// TwinCAT 3 PLC project PRG_B_Base
// Title: B_Base
// Company: RafalOS
// Author: Rafał Osajda
// ProjectVersion: 0.0.1.0
// ProgramVersion: 3.1.4024.0
// libraries:
//   Tc2_Standard, * (Beckhoff Automation GmbH)
//   Tc2_System, * (Beckhoff Automation GmbH)
//   Tc2_Utilities, * (Beckhoff Automation GmbH)
//   Tc3_Module, * (Beckhoff Automation GmbH)
// project tree:
//   DUTs Events/ E_BaseEvents_Category.TcDUT, E_BaseEvents_Action.TcDUT (not stored), ST_BaseEvents.TcDUT (not stored), ST_BaseEvents_ActiveEvents.TcDUT (not stored), ST_BaseEvents_Definition.TcDUT, ST_BaseEvents_Queue.TcDUT, ST_BaseEvents_Memory.TcDUT, ST_BaseEvents_RowInQueue.TcDUT (not stored), ST_BaseEvents_RowInMemory.TcDUT (not stored), ST_BaseEvents_InformationAboutEventsForHMI.TcDUT
//   DUTs/ E_BaseElementType.TcDUT (not stored), E_BaseLocation.TcDUT (not stored), E_BaseMachineState.TcDUT (not stored), E_BaseMachineMode.TcDUT (not stored), ST_BaseCommonData.TcDUT, ST_BaseDescriptor.TcDUT, ST_BaseElementIdentifier.TcDUT (not stored), ST_BaseLocationDesctription.TcDUT, ST_BaseLabel.TcDUT
//   FUNs/ CreateElementCode.TcPOU
//   GVLs/ GVL_BaseConstans.TcGVL (not stored)
//   ITFs/ ITF_DecoratedElement.TcIO (not stored)
//   / PlcTask.TcTTO
//   POUs Compilation/ PRG_Compilation.TcPOU
//   POUs/A01_Base/ ITF_Base.TcIO, FB_Base.TcPOU (not stored)
//   POUs/A02_FB_BaseLogger/ ITF_BaseLogger_HMI_Connector.TcIO, ITF_BaseLogger_HMI_Connector_Command.TcIO, FB_BaseLogger.TcPOU (not stored), ITF_BaseLogger.TcIO, ITF_BaseLogger_HMI_Connector_View.TcIO, ITF_BaseLogger_Item.TcIO, ST_BaseLogger_ItemDataToDisplay.TcDUT
//   POUs/A03_FB_BaseLoggerElement/ ITF_BaseLoggerElement_HMI_Connector.TcIO, ITF_BaseLoggerElement_HMI_Connector_Command.TcIO, FB_BaseLoggerElement.TcPOU, ITF_BaseLoggerElement.TcIO, ITF_BaseLoggerElement_HMI_Connector_View.TcIO
//   POUs/A04_FB_BaseComponent/ ITF_BaseComponent_HMI_Connector.TcIO, ITF_BaseComponent_HMI_Connector_Command.TcIO, FB_BaseComponent.TcPOU, ITF_BaseComponent.TcIO, ITF_BaseComponent_HMI_Connector_View.TcIO, ST_Parameters.TcDUT
//   POUs/A05_FB_BaseControlElement/ ITF_BaseControlElement_HMI_Connector.TcIO, ITF_BaseControlElement_HMI_Connector_Command.TcIO, FB_BaseControlElement.TcPOU, ITF_BaseControlElement.TcIO, ITF_BaseControlElement_HMI_Connector_View.TcIO, ST_BaseControlElement_Power.TcDUT, ST_BaseControlElement_Homing.TcDUT (not stored)
//   POUs/A06_FB_BaseGroupElement/ ITF_BaseGroupElement_HMI_Connector.TcIO, ITF_BaseGroupElement_HMI_Connector_Command.TcIO, FB_BaseGroupElement.TcPOU, ITF_BaseGroupElement.TcIO (not stored), ITF_BaseGroupElement_HMI_Connector_View.TcIO
//   POUs/A07_FB_BaseTopElement/ ITF_BaseSaM.TcIO, ITF_BaseSaMStateMethod.TcIO (not stored), ITF_BaseTopElement_HMI_Connector.TcIO, ITF_BaseTopElement_HMI_Connector_Command.TcIO, FB_BaseTopElement.TcPOU (not stored), ITF_BaseTopElement.TcIO (not stored), ITF_BaseTopElement_HMI_Connector_View.TcIO
//   POUs/B01_Komunikator/ ITF_BaseCommunicator.TcIO, ITF_BaseMessengerRecipient.TcIO, ITF_BaseMessengerSender.TcIO (not stored), FB_BaseCommunicator.TcPOU (not stored), ST_BaseCommunicatorData.TcDUT, ST_BaseCommunicatorStack.TcDUT, ST_BaseCommunicatorMassege.TcDUT (not stored)
//   POUs/B02_Recipes/ FB_BaseRecipe.TcPOU, ITF_BaseCreateTemplateOfRecipe.TcIO (not stored), ITF_BaseCreatingTemplateMethod.TcIO, ITF_BaseRecipe.TcIO, ITF_BaseRecipe_HMI_Connector.TcIO, ST_BaseRecipeListRow.TcDUT, ST_BaseRecipe.TcDUT (not stored), ST_BaseRecipeList.TcDUT
//   POUs/A00_Basic/ FB_BaseLabel.TcPOU, FB_BaseTime.TcPOU (not stored), FB_BaseCommand.TcPOU (not stored), FB_BaseDescriptor.TcPOU, FB_BaseFlag.TcPOU, FB_BaseImpulse.TcPOU (not stored), FB_BaseLocation.TcPOU (not stored), ITF_BaseDescriptor.TcIO, ITF_BaseFlag.TcIO (not stored), ITF_BaseFlagGet.TcIO, ITF_BaseFlagSet.TcIO (not stored), ITF_BaseImpulse.TcIO (not stored), ITF_BaseLabel.TcIO, ITF_BaseLocation.TcIO, ITF_BaseTime.TcIO

CONFIGURATION PRG_B_Base
    RESOURCE PLC ON TwinCAT3
        TASK PlcTask(INTERVAL := T#10ms, PRIORITY := 20);
        PROGRAM PRG_Compilation WITH PlcTask : PRG_Compilation;
    END_RESOURCE
END_CONFIGURATION

// ---- DUTs Events/E_BaseEvents_Category.TcDUT
{attribute 'qualified_only'}
{attribute 'strict'}
{attribute 'to_string'}
TYPE E_BaseEvents_Category :
(
	None		:= 0,
	Error		:= 1, 
	Alarm		:= 2, 
	Safety		:= 3, 
	Message		:= 4

);
END_TYPE

// ---- DUTs Events/ST_BaseEvents_Definition.TcDUT
TYPE ST_BaseEvents_Definition :
STRUCT
	uiIDEvent								: UINT;						//unikalny numer zgloszenia dla całego projektu nadawany automatycznie 
	uiIDInItem								: UINT;						//unikalny numer w elemencie - ustawiany podczas dodawania zgłoszenia DO elementu
	bIgnoreRepetitions						: BOOL;						//jak true nie zliczaj powtorzeń wystapienia np komunikaty - alarmy 
	uiRepetitionCounter						: UINT;						//licznik powtórzeń po którym ma się zgłosic błąd
	eEventCategory							: E_BaseEvents_Category;	//BYTE;	//1 - blad, 2 - ostrzezenie, 3 - wiadomosc, 4 - safety
	stDescription							: ST_BaseLabel;
	bConfirm								: BOOL;						// w przypadków niektórych zgłoszeń żeby błąd został skasowany należy go zatwierdzić że operator go zobaczył
END_STRUCT
END_TYPE

// ---- DUTs Events/ST_BaseEvents_Queue.TcDUT
TYPE ST_BaseEvents_Queue :
STRUCT
	arrEvents						: ARRAY [1..GVL_BaseConstans.MAX_NUMBER_OF_EVENTS_IN_THE_QUEUE] OF ST_BaseEvents_RowInQueue;
	iNumerOfEvents					: INT;

END_STRUCT
END_TYPE

// ---- DUTs Events/ST_BaseEvents_Memory.TcDUT
TYPE ST_BaseEvents_Memory :
STRUCT
	arrRow						: ARRAY [1..GVL_BaseConstans.MAX_EVENTS_IN_MEMORY] OF ST_BaseEvents_RowInMemory;
	iNumberOfRow				: INT;
	
END_STRUCT
END_TYPE

// ---- DUTs Events/ST_BaseEvents_InformationAboutEventsForHMI.TcDUT
(*			
	RafalOS
	Rafał Osajda		03.09.2025		TC 4024.66
	Informacja czy w danym elemencie jest jakieś nowe zgłoszenie jeszcze nei wyświetlane i ilosc zgloszen calkowita
*)
TYPE ST_BaseEvents_InformationAboutEventsForHMI :
STRUCT
	bNew				: BOOL;	//nowe
	iQuantity			: INT;	//Ilość
END_STRUCT
END_TYPE

// ---- DUTs/ST_BaseCommonData.TcDUT
TYPE ST_BaseCommonData :
STRUCT
	itfLogger				: ITF_BaseLogger;
	itfTime					: ITF_BaseTime;
	itfLocaciotn			: ITF_BaseLocation;
END_STRUCT
END_TYPE

// ---- DUTs/ST_BaseDescriptor.TcDUT
TYPE ST_BaseDescriptor :
STRUCT
	stTexts						: ST_BaseLabel;
	sUnit						: STRING(6);
	rValue						: REAL;
	rMin						: REAL;
	rMax						: REAL;
	rDefaultValue				: REAL;
	
END_STRUCT
END_TYPE

// ---- DUTs/ST_BaseLocationDesctription.TcDUT
TYPE ST_BaseLocationDesctription :
STRUCT
	wsDescription		: WSTRING;
	sCode				: STRING(5);
END_STRUCT
END_TYPE

// ---- DUTs/ST_BaseLabel.TcDUT
TYPE ST_BaseLabel :
STRUCT
	arrText		: ARRAY [1..GVL_BaseConstans.NUMBER_OF_LOCATIONS] OF WSTRING;
	
END_STRUCT
END_TYPE

// ---- POUs/B01_Komunikator/ST_BaseCommunicatorData.TcDUT
TYPE ST_BaseCommunicatorData :
STRUCT
	stMessage					: ST_BaseCommunicatorMassege;
	itfSender					: ITF_BaseMessengerSender;
	arritfRecipient				: ARRAY [1..GVL_BaseConstans.MAX_NUMBER_OF_CLIENTS] OF ITF_BaseMessengerRecipient;
	arrConfirmations			: ARRAY [1..GVL_BaseConstans.MAX_NUMBER_OF_CLIENTS] OF BOOL;		//potwierdzenia
	iNumberOfConfirmations		: INT;	//ilosc odbiorcow ktorzy musza potwierdzic
	iNumberOfRecipient			: INT;
END_STRUCT
END_TYPE

// ---- POUs/B01_Komunikator/ST_BaseCommunicatorStack.TcDUT
TYPE ST_BaseCommunicatorStack :
STRUCT
	stMessage					: ST_BaseCommunicatorMassege;
	bSent						: BOOL;		//wysłane
	bConfirmation				: BOOL;		//potwierdzenie
	itfSender					: ITF_BaseMessengerSender;
	itfRecipient				: ITF_BaseMessengerRecipient;
	
END_STRUCT
END_TYPE

// ---- POUs/A02_FB_BaseLogger/ST_BaseLogger_ItemDataToDisplay.TcDUT
TYPE ST_BaseLogger_ItemDataToDisplay :
STRUCT
	sCode						: STRING;
	sEventCategory				: STRING;
	eEventCategory				: E_BaseEvents_Category;
	stDescription				: ST_BaseLabel;
	stItemName					: ST_BaseLabel;
	uiRepetitionCounter			: UINT;
END_STRUCT
END_TYPE

// ---- POUs/A04_FB_BaseComponent/ST_Parameters.TcDUT
TYPE ST_Parameters :
STRUCT
	arrRow	 				: ARRAY [1..GVL_BaseConstans.MAX_NUMBER_OF_PARAMETERS] OF ST_BaseDescriptor;
	uiNumber				: UINT;
END_STRUCT
END_TYPE

// ---- POUs/A05_FB_BaseControlElement/ST_BaseControlElement_Power.TcDUT
TYPE ST_BaseControlElement_Power :
STRUCT
	cmdTurnOn				: FB_BaseCommand;
	cmdTurnOff				: FB_BaseCommand;
	bStatus					: BOOL;
END_STRUCT
END_TYPE

// ---- POUs/B02_Recipes/ST_BaseRecipeListRow.TcDUT
TYPE ST_BaseRecipeListRow :
STRUCT
	wsText			: WSTRING;
	iNumber			: INT;
	refRecipe		: REFERENCE TO ST_BaseRecipe;
END_STRUCT
END_TYPE

// ---- POUs/B02_Recipes/ST_BaseRecipeList.TcDUT
TYPE ST_BaseRecipeList :
STRUCT
	arrName 	: ARRAY [1..GVL_BaseConstans.MAX_NUMBER_OF_RECIPES] OF ST_BaseLabel;
	iNumber		: INT;
END_STRUCT
END_TYPE

// ---- POUs/A01_Base/ITF_Base.TcIO
INTERFACE ITF_Base

METHOD PUBLIC SetName
VAR_INPUT
	stName				: ST_BaseLabel;
END_VAR
END_METHOD

END_INTERFACE

// ---- POUs/A02_FB_BaseLogger/ITF_BaseLogger_HMI_Connector.TcIO
INTERFACE ITF_BaseLogger_HMI_Connector EXTENDS ITF_BaseLogger_HMI_Connector_Command, ITF_BaseLogger_HMI_Connector_View

END_INTERFACE

// ---- POUs/A02_FB_BaseLogger/ITF_BaseLogger_HMI_Connector_Command.TcIO
INTERFACE ITF_BaseLogger_HMI_Connector_Command

END_INTERFACE

// ---- POUs/A03_FB_BaseLoggerElement/ITF_BaseLoggerElement_HMI_Connector.TcIO
INTERFACE ITF_BaseLoggerElement_HMI_Connector EXTENDS
		ITF_BaseLoggerElement_HMI_Connector_Command, ITF_BaseLoggerElement_HMI_Connector_View

END_INTERFACE

// ---- POUs/A03_FB_BaseLoggerElement/ITF_BaseLoggerElement_HMI_Connector_Command.TcIO
INTERFACE ITF_BaseLoggerElement_HMI_Connector_Command

END_INTERFACE

// ---- POUs/A04_FB_BaseComponent/ITF_BaseComponent_HMI_Connector.TcIO
INTERFACE ITF_BaseComponent_HMI_Connector EXTENDS ITF_BaseComponent_HMI_Connector_View, ITF_BaseComponent_HMI_Connector_Command

END_INTERFACE

// ---- POUs/A04_FB_BaseComponent/ITF_BaseComponent_HMI_Connector_Command.TcIO
INTERFACE ITF_BaseComponent_HMI_Connector_Command

END_INTERFACE

// ---- POUs/A05_FB_BaseControlElement/ITF_BaseControlElement_HMI_Connector.TcIO
INTERFACE ITF_BaseControlElement_HMI_Connector EXTENDS 
		ITF_BaseControlElement_HMI_Connector_View, ITF_BaseControlElement_HMI_Connector_Command

END_INTERFACE

// ---- POUs/A05_FB_BaseControlElement/ITF_BaseControlElement_HMI_Connector_Command.TcIO
INTERFACE ITF_BaseControlElement_HMI_Connector_Command

END_INTERFACE

// ---- POUs/A06_FB_BaseGroupElement/ITF_BaseGroupElement_HMI_Connector.TcIO
INTERFACE ITF_BaseGroupElement_HMI_Connector EXTENDS 
		ITF_BaseGroupElement_HMI_Connector_View, ITF_BaseGroupElement_HMI_Connector_Command

END_INTERFACE

// ---- POUs/A06_FB_BaseGroupElement/ITF_BaseGroupElement_HMI_Connector_Command.TcIO
INTERFACE ITF_BaseGroupElement_HMI_Connector_Command

END_INTERFACE

// ---- POUs/A07_FB_BaseTopElement/ITF_BaseSaM.TcIO
INTERFACE ITF_BaseSaM

METHOD PUBLIC GetMode : E_BaseMachineMode
VAR_INPUT
END_VAR
END_METHOD

METHOD PUBLIC GetState : E_BaseMachineState
VAR_INPUT
END_VAR
END_METHOD

(*			
	RafalOS
	Rafał Osajda		25.10.2025		TC 4024.66
	Czy trwa zmianay trybu
*)
METHOD PUBLIC IsChangeModeBusy : BOOL
VAR_INPUT
END_VAR
END_METHOD

(*			
	RafalOS
	Rafał Osajda		25.10.2025		TC 4024.66
	Czy trwa zmiana stanu
*)
METHOD PUBLIC IsChangeStateBusy : BOOL
VAR_INPUT

END_VAR
END_METHOD

END_INTERFACE

// ---- POUs/A07_FB_BaseTopElement/ITF_BaseTopElement_HMI_Connector.TcIO
INTERFACE ITF_BaseTopElement_HMI_Connector EXTENDS ITF_BaseTopElement_HMI_Connector_View, ITF_BaseTopElement_HMI_Connector_Command

END_INTERFACE

// ---- POUs/A07_FB_BaseTopElement/ITF_BaseTopElement_HMI_Connector_Command.TcIO
INTERFACE ITF_BaseTopElement_HMI_Connector_Command

END_INTERFACE

// ---- POUs/B01_Komunikator/ITF_BaseCommunicator.TcIO
INTERFACE ITF_BaseCommunicator

METHOD PUBLIC ReceiveData_BOOL : BOOL
VAR_INPUT
	sText			: STRING;
	itfRecipient	: ITF_BaseMessengerRecipient;
END_VAR
VAR_OUTPUT
	bValue			: BOOL;	
END_VAR
END_METHOD

METHOD PUBLIC ReceiveData_REAL : BOOL
VAR_INPUT
	sText			: STRING;
	itfRecipient	: ITF_BaseMessengerRecipient;
END_VAR
VAR_OUTPUT
	rValue			: REAL;	
END_VAR
END_METHOD

(*			
	RafalOS
	Rafał Osajda		30.07.2025		TC 4024.66
	Wysyła potwierdzenie że odebrał dane
*)
METHOD PUBLIC ReceiveDataConfirm : BOOL
VAR_INPUT
	sText				: STRING;
	itfRecipient		: ITF_BaseMessengerRecipient;
END_VAR
END_METHOD

METHOD SendData_BOOL : BOOL
VAR_INPUT
	sText		: STRING;
	itfSender	: ITF_BaseMessengerSender;
END_VAR
END_METHOD

METHOD SendData_REAL : BOOL
VAR_INPUT
	sText		: STRING;
	rValue		: REAL;
	itfSender	: ITF_BaseMessengerSender;
END_VAR
END_METHOD

END_INTERFACE

// ---- POUs/B01_Komunikator/ITF_BaseMessengerRecipient.TcIO
INTERFACE ITF_BaseMessengerRecipient

END_INTERFACE

// ---- POUs/A00_Basic/ITF_BaseDescriptor.TcIO
INTERFACE ITF_BaseDescriptor

METHOD PUBLIC GetDefaultValue : REAL
VAR_INPUT
END_VAR
END_METHOD

METHOD PUBLIC GetMax : REAL
VAR_INPUT
END_VAR
END_METHOD

METHOD PUBLIC GetMin : REAL
VAR_INPUT
END_VAR
END_METHOD

METHOD PUBLIC GetTexts : ST_BaseLabel
VAR_INPUT
END_VAR
END_METHOD

METHOD PUBLIC GetUnit : STRING(6)
VAR_INPUT
END_VAR
END_METHOD

METHOD PUBLIC GetValue : REAL
VAR_INPUT
END_VAR
END_METHOD

METHOD PUBLIC SetDefaultValue
VAR_INPUT
	rDefaultValue: REAL;
END_VAR
END_METHOD

METHOD PUBLIC SetMax
VAR_INPUT
	rMax: REAL;
END_VAR
END_METHOD

METHOD PUBLIC SetMin
VAR_INPUT
	rMin: REAL;
END_VAR
END_METHOD

METHOD PUBLIC SetText
VAR_INPUT
	eLocation			: E_BaseLocation;
	wsDescription		: WSTRING;
END_VAR
END_METHOD

METHOD PUBLIC SetTexts
VAR_INPUT
	stTexts				: ST_BaseLabel;
END_VAR
END_METHOD

METHOD PUBLIC SetUnit
VAR_INPUT
	sUnit: STRING(6);
END_VAR
END_METHOD

METHOD PUBLIC SetValue
VAR_INPUT
	rValue: REAL;
END_VAR
END_METHOD

END_INTERFACE

// ---- POUs/A00_Basic/ITF_BaseFlagGet.TcIO
INTERFACE ITF_BaseFlagGet

METHOD PUBLIC GetFlag : BOOL
VAR_INPUT
END_VAR
END_METHOD

END_INTERFACE

// ---- POUs/A00_Basic/ITF_BaseLabel.TcIO
INTERFACE ITF_BaseLabel

METHOD PUBLIC GetTexts : ST_BaseLabel
VAR_INPUT
END_VAR
END_METHOD

METHOD PUBLIC SetText
VAR_INPUT
	eLocation			: E_BaseLocation;
	wsDescription		: WSTRING;
END_VAR
END_METHOD

METHOD PUBLIC SetTexts
VAR_INPUT
	stTexts				: ST_BaseLabel;
END_VAR
END_METHOD

END_INTERFACE

// ---- POUs/A00_Basic/ITF_BaseLocation.TcIO
INTERFACE ITF_BaseLocation

(*			
	RAFALOS
	Rafał Osajda		24.09.2025		TC 4024.66
	Zwraca kod jezyka tzn 
*)
METHOD PUBLIC GetActualCode : STRING
VAR_INPUT
END_VAR
END_METHOD

METHOD PUBLIC GetActualDescription : WSTRING
VAR_INPUT
END_VAR
END_METHOD

METHOD PUBLIC GetCode : STRING(5)
VAR_INPUT
	iIN				: INT;
END_VAR
END_METHOD

METHOD PUBLIC GetDescription : WSTRING
VAR_INPUT
	iIN				: INT;
END_VAR
END_METHOD

METHOD PUBLIC GetLocation : E_BaseLocation
VAR_INPUT
END_VAR
END_METHOD

METHOD PUBLIC SetLocation : BOOL
VAR_INPUT
	sLocation				: STRING;
END_VAR
END_METHOD

END_INTERFACE

// ---- POUs/A00_Basic/ITF_BaseTime.TcIO
INTERFACE ITF_BaseTime

(*			
	RafalOS
	Rafał Osajda		01.09.2025		TC 4024.66
	Konwetrtuje DT to string do postaci DD/MM/YYYY GG:MM:SS
*)
METHOD PUBLIC BaseDTToString : STRING
VAR_INPUT
	inDT					: DT;
END_VAR
END_METHOD

(*			
	RafalOS
	Rafał Osajda		01.09.2025		TC 4024.66
	Konwetrtuje DT to string do postaci DD_MM_YYYY GG_MM_SS - wersja do nazywania plików logów
*)
METHOD PUBLIC BaseDTToString_ : STRING
VAR_INPUT
	inDT				: DT;
END_VAR
END_METHOD

(*			
	RafalOS
	Rafał Osajda		01.09.2025		TC 4024.66
	Konwertuje czas LTIME do stringa z możliwością wyłączenia milisekund
*)
METHOD PUBLIC BaseLTimeToString : STRING
VAR_INPUT
	ltTime				: LTIME;
	bShowMS			: BOOL;
END_VAR
END_METHOD

(*			
	RafalOS
	Rafał Osajda		01.09.2025		TC 4024.66
	Konwertuje czas LTIME do stringa z możliwością wybrnia co ma być pokazywane do postaci DDDd:GG:MM:SS:MS
	dni nie rodziala na miesiące i lata 
*)
METHOD PUBLIC BaseLTimeToString_WhatShow : STRING
VAR_INPUT
	ltTime				: LTIME;
	bSwahDays			: BOOL;
	bShowHours			: BOOL;
	bShowMinutes		: BOOL;
	bShowSeconds		: BOOL;
	bShowMS				: BOOL;
END_VAR
END_METHOD

METHOD PUBLIC StampDT : DT
VAR_INPUT
END_VAR
END_METHOD

END_INTERFACE

// ---- POUs/A02_FB_BaseLogger/ITF_BaseLogger.TcIO
INTERFACE ITF_BaseLogger

METHOD PUBLIC AddItem : INT
VAR_INPUT
	itfItem				: ITF_BaseLogger_Item;
END_VAR
END_METHOD

METHOD PUBLIC GetNumerOfReportsIntheSystem : UINT
VAR_INPUT
END_VAR
END_METHOD

METHOD PUBLIC ReportEvent : BOOL
VAR_INPUT
	stEvent					: ST_BaseEvents_RowInQueue;
END_VAR
END_METHOD

METHOD PUBLIC SetNumerOfReportsIntheSystem
VAR_INPUT
	uiValue		: UINT;
END_VAR
END_METHOD

END_INTERFACE

// ---- POUs/A02_FB_BaseLogger/ITF_BaseLogger_HMI_Connector_View.TcIO
INTERFACE ITF_BaseLogger_HMI_Connector_View

(*			
	RafalOS
	Rafał Osajda		02.10.2025		TC 4024.66
	Zwraca czy nastąpiła jakaś zmiana w pamięci zgłoszeń - całej nie tylko dla jakiegoś elementu
*)
METHOD PUBLIC GetChangeInMemory : BOOL
VAR_INPUT
END_VAR
END_METHOD

METHOD PUBLIC GetEventCounts : ST_BaseEvents_ActiveEvents
VAR_INPUT
END_VAR
END_METHOD

METHOD PUBLIC GetEventCountsForItem : ST_BaseEvents_ActiveEvents
VAR_INPUT
	uiIDItem: UINT;
END_VAR
END_METHOD

METHOD PUBLIC GetInformationFromItem : ST_BaseLogger_ItemDataToDisplay
VAR_INPUT
	uiIDItem				: UINT;
	uiIDEvent				: UINT;
END_VAR
END_METHOD

METHOD GetReferenceToStmemory : REFERENCE TO ST_BaseEvents_Memory
VAR_INPUT
	
END_VAR
END_METHOD

(*			
	RafalOS
	Rafał Osajda		02.10.2025		TC 4024.66
	
*)
METHOD PUBLIC ResetChangeInMemory : BOOL
VAR_INPUT
END_VAR
END_METHOD

END_INTERFACE

// ---- POUs/A02_FB_BaseLogger/ITF_BaseLogger_Item.TcIO
INTERFACE ITF_BaseLogger_Item

METHOD PUBLIC GetID : UINT
VAR_INPUT
END_VAR
END_METHOD

METHOD GetInformationToDisplayEvent : ST_BaseLogger_ItemDataToDisplay
VAR_INPUT
	uiIDEvent				: UINT;
END_VAR
END_METHOD

END_INTERFACE

// ---- POUs/A03_FB_BaseLoggerElement/ITF_BaseLoggerElement.TcIO
INTERFACE ITF_BaseLoggerElement EXTENDS ITF_Base

(*			
	RafalOS
	Rafał Osajda		24.03.2025		TC 4024.66
	Definicja nowego zgłoszenia
*)
METHOD PUBLIC EventsDefinition : BOOL
END_METHOD

METHOD PUBLIC GetCode : STRING
VAR_INPUT
END_VAR
END_METHOD

METHOD PUBLIC GetID : UINT
VAR_INPUT
END_VAR
END_METHOD

METHOD PUBLIC GetIdentyfier : ST_BaseElementIdentifier
VAR_INPUT
END_VAR
END_METHOD

METHOD PUBLIC GetName : ST_BaseLabel
VAR_INPUT
END_VAR
END_METHOD

METHOD PUBLIC GetType : E_BaseElementType
VAR_INPUT
END_VAR
END_METHOD

METHOD PUBLIC SetCode
VAR_INPUT
	sCode							: STRING;
	sAdd							: STRING;
END_VAR
END_METHOD

(*			
	RafalOS
	Rafał Osajda		03.10.2025		TC 4024.66
	nadawanie unikalnych ID dla zdarzeń
*)
METHOD PUBLIC SetEventsIDs : UINT
VAR_INPUT
	uiNewID		: UINT;
END_VAR
END_METHOD

METHOD PUBLIC SetID : UINT
VAR_INPUT
	uiID					: UINT;
END_VAR
END_METHOD

METHOD PUBLIC SetName
VAR_INPUT
	stName				: ST_BaseLabel;
END_VAR
END_METHOD

METHOD PUBLIC SetType
VAR_INPUT
	eType					: E_BaseElementType;
END_VAR
END_METHOD

END_INTERFACE

// ---- POUs/A03_FB_BaseLoggerElement/ITF_BaseLoggerElement_HMI_Connector_View.TcIO
INTERFACE ITF_BaseLoggerElement_HMI_Connector_View

(*			
	RafalOS
	Rafał Osajda		09.06.2025		TC 4024.66
	Szuka czy ma zgłoszenie i zadanym ID jak tak to usuwa i zwraca true w przeciwnym razie zwraca false 
*)
METHOD PUBLIC EventAcknowledgeByID : BOOL
VAR_INPUT
	uiIDEvent				: UINT;
END_VAR
END_METHOD

(*			
	RafalOS
	Rafał Osajda		09.06.2025		TC 4024.66
	Szuka czy ma zgłoszenie i zadanym ID jak tak to usuwa i zwraca true w przeciwnym razie zwraca false 
*)
METHOD PUBLIC EventSetInactiveByID : BOOL
VAR_INPUT
	uiIDEvent				: UINT;
END_VAR
END_METHOD

METHOD PUBLIC GetCode : STRING
VAR_INPUT
END_VAR
END_METHOD

METHOD PUBLIC GetID : UINT
VAR_INPUT
END_VAR
END_METHOD

METHOD PUBLIC GetIdentyfier : ST_BaseElementIdentifier
VAR_INPUT
END_VAR
END_METHOD

METHOD PUBLIC GetName : ST_BaseLabel
VAR_INPUT
END_VAR
END_METHOD

METHOD PUBLIC GetType : E_BaseElementType
VAR_INPUT
END_VAR
END_METHOD

END_INTERFACE

// ---- POUs/A04_FB_BaseComponent/ITF_BaseComponent.TcIO
INTERFACE ITF_BaseComponent EXTENDS ITF_BaseLoggerElement

(*			
	RafalOS
	Rafał Osajda		27.03.2025		TC 4024.66
	Obsluga bledow sprawdzanie czy jakis blad sie nei pojawil i ustawienie stanu lub wylaczenie
*)
METHOD PUBLIC ExecuteEveryCycle_Error
VAR_INPUT
END_VAR
END_METHOD

(*			
	RafalOS
	Rafał Osajda		27.03.2025		TC 4024.66
	Wywolanie co cykl operacji 
*)
METHOD PUBLIC ExecuteEveryCycle_Operation
VAR_INPUT
END_VAR
END_METHOD

(*			
	RafalOS
	Rafał Osajda		27.03.2025		TC 4024.66
	Aktualizacja flag 
*)
METHOD PUBLIC ExecuteEveryCycle_Status
VAR_INST
END_VAR
END_METHOD

(*			
	RafalOS
	Rafał Osajda		27.03.2025		TC 4024.66
	Testowanie czy nei pojawil sie jakis rozkaz i uruchomienie odpowiednich operacji
*)
METHOD PUBLIC ExecuteEveryCycle_Test
VAR_INPUT
END_VAR
END_METHOD

METHOD PUBLIC FirstCycle : BOOL
VAR_INPUT
END_VAR
END_METHOD

METHOD PUBLIC IsValidCommonData : BOOL
VAR_INPUT
END_VAR
END_METHOD

(*			
	RafalOS
	Rafał Osajda		07.10.2025		TC 4024.66
	Dodpisywanie się do listy logera
*)
METHOD PUBLIC JoinTheLogger : BOOL
VAR_INPUT
END_VAR
END_METHOD

METHOD PUBLIC LinkCommonData : BOOL
VAR_INPUT
	stCommonData				: REFERENCE TO ST_BaseCommonData;
END_VAR
END_METHOD

(*			
	RafalOS
	Rafał Osajda		26.03.2025		TC 4024.66
	Dodawanie parametru do elementu wykonawczego - metode wywołać przy pierwszym uruchomieniu programu by wgrać parametry do pamięci
	później używać tylko edycji lub przywracania wartości domyślnych
*)
METHOD PUBLIC ParameterAdd : BOOL
VAR_INPUT
	stParameter			: ST_BaseDescriptor;
END_VAR
END_METHOD

(*			
	RafalOS
	Rafał Osajda		26.03.2025		TC 4024.66
	Modyfikuje wartość domyślną w istniejącym parametrze - true jak się zmiana udała
*)
METHOD PUBLIC ParameterCorrectDefaultValue : BOOL
VAR_INPUT
	uiNumber			: UINT;
	rValue				: REAL;
END_VAR
END_METHOD

METHOD PUBLIC ParameterCorrectName : BOOL
VAR_INPUT
	eLocation					: E_BaseLocation;
	uiNumberOfParameter			: UINT;
	wsDescription				: WSTRING;
END_VAR
END_METHOD

(*			
	RafalOS
	Rafał Osajda		26.03.2025		TC 4024.66
	Modyfikuje wartość w istniejącym parametrze - true jak się zmiana udała
*)
METHOD PUBLIC ParameterCorrectValue : BOOL
VAR_INPUT
	uiNumber			: UINT;
	rValue				: REAL;
END_VAR
END_METHOD

METHOD PUBLIC ParameterGet : ST_BaseDescriptor
VAR_INPUT
	uiNumer				: UINT;
END_VAR
END_METHOD

(*			
	RafalOS
	Rafał Osajda		26.03.2025		TC 4024.66
	Zwraca wartosc domyslna
*)
METHOD PUBLIC ParameterGetDefaultValue : REAL
VAR_INPUT
	uiNumber				: UINT;
END_VAR
END_METHOD

(*			
	RafalOS
	Rafał Osajda		26.03.2025		TC 4024.66
	Zwraca wartość MAX
*)
METHOD PUBLIC ParameterGetMax : REAL
VAR_INPUT
	uiNumber				: UINT;
END_VAR
END_METHOD

(*			
	RafalOS
	Rafał Osajda		26.03.2025		TC 4024.66
	Zwraca wartość MIN
*)
METHOD PUBLIC ParameterGetMin : REAL
VAR_INPUT
	uiNumber				: UINT;
END_VAR
END_METHOD

METHOD PUBLIC ParameterGetNumberOfAdded : UINT
VAR_INPUT
END_VAR
END_METHOD

(*			
	RafalOS
	Rafał Osajda		26.03.2025		TC 4024.66
	Zwraca jednostke
*)
METHOD PUBLIC ParameterGetUnit : STRING(6)
VAR_INPUT
	uiNumber				: uINT;
END_VAR
END_METHOD

(*			
	RafalOS
	Rafał Osajda		26.03.2025		TC 4024.66
	Zwraca wartość
*)
METHOD PUBLIC ParameterGetValue : REAL
VAR_INPUT
	uiNumber				: UINT;
END_VAR
END_METHOD

(*			
	RafalOS
	Rafał Osajda		26.03.2025		TC 4024.66
	Modyfikacja istniejącego parametra jako przypisanie nowego deskryptora
*)
METHOD PUBLIC ParameterModify : BOOL
VAR_INPUT
	uiNumber			: UINT;
	stParameter			: ST_BaseDescriptor;
END_VAR
END_METHOD

METHOD PUBLIC ParameterRestoreDefaultValue : BOOL
VAR_INPUT
	uiNumber		: UINT;
END_VAR
END_METHOD

(*			
	RafalOS
	Rafał Osajda		04.05.2025		TC 4024.66
	Skasowanie i utworzenie tablicy parametrów od nowa 
*)
METHOD PUBLIC ParametersCreate : BOOL
END_METHOD

(*			
	RafalOS
	Rafał Osajda		04.05.2025		TC 4024.66
	Przywrocenie parametrow - in na false to tylko ten element true razem z podelementami
*)
METHOD PUBLIC ParameterSetToDefault : BOOL
END_METHOD

METHOD PUBLIC Reset : BOOL
VAR_INPUT
END_VAR
END_METHOD

METHOD PUBLIC ResetGetBusy : BOOL
VAR_INPUT
END_VAR
END_METHOD

METHOD PUBLIC ResetGetStatus : BOOL
VAR_INPUT
END_VAR
END_METHOD

END_INTERFACE

// ---- POUs/A04_FB_BaseComponent/ITF_BaseComponent_HMI_Connector_View.TcIO
INTERFACE ITF_BaseComponent_HMI_Connector_View EXTENDS ITF_BaseLoggerElement_HMI_Connector_View

END_INTERFACE

// ---- POUs/A05_FB_BaseControlElement/ITF_BaseControlElement.TcIO
INTERFACE ITF_BaseControlElement EXTENDS ITF_BaseComponent

(*			
	RafalOS
	Rafał Osajda		31.03.2025		TC 4024.66
	Flaga że w tej sesji pracy maszyny element został już wybazowany
*)
METHOD PUBLIC HomingGetDone : BOOL
VAR_INPUT
END_VAR
END_METHOD

(*			
	RafalOS
	Rafał Osajda		11.04.2025		TC 4024.66
	Zwraca czy bazowanie jest potrzebne
*)
METHOD PUBLIC HomingGetIsNeeded : BOOL
VAR_INPUT
END_VAR
END_METHOD

(*			
	RafalOS
	Rafał Osajda		27.05.2025		TC 4024.66
	Uruchomienie metody bazowania
*)
METHOD PUBLIC HomingStart
VAR_INPUT
END_VAR
END_METHOD

(*			
	RafalOS
	Rafał Osajda		30.04.2025		TC 4024.66
	Zwraca czy element jest czymś zajety
*)
METHOD PUBLIC IsDoNothing : BOOL
END_METHOD

(*			
	RafalOS
	Rafał Osajda		30.04.2025		TC 4024.66
	Zwraca czy element jest w pozycji 0 - referencyjnej
*)
METHOD PUBLIC IsPosition0 : BOOL
END_METHOD

METHOD PUBLIC LinkSS1 : BOOL
VAR_INPUT
	fbSS1			: ITF_BaseFlagGet;
END_VAR
END_METHOD

METHOD PUBLIC LinkSTO : BOOL
VAR_INPUT
	fbSTO			: ITF_BaseFlagGet;
END_VAR
END_METHOD

(*			
	RafalOS
	Rafał Osajda		31.03.2025		TC 4024.66
	Zwraca status zasilania	
*)
METHOD PUBLIC PowerGetStatus : BOOL
VAR_INPUT
END_VAR
END_METHOD

(*			
	RafalOS
	Rafał Osajda		31.03.2025		TC 4024.66
	Wyłączenie zasilania
*)
METHOD PUBLIC PowerTurnOff : BOOL
VAR_INPUT
END_VAR
END_METHOD

(*			
	RafalOS
	Rafał Osajda		31.03.2025		TC 4024.66
	Uruchomienie zasialania
*)
METHOD PUBLIC PowerTurnOn
VAR_INPUT
END_VAR
END_METHOD

END_INTERFACE

// ---- POUs/A05_FB_BaseControlElement/ITF_BaseControlElement_HMI_Connector_View.TcIO
INTERFACE ITF_BaseControlElement_HMI_Connector_View EXTENDS ITF_BaseComponent_HMI_Connector_View

END_INTERFACE

// ---- POUs/A06_FB_BaseGroupElement/ITF_BaseGroupElement_HMI_Connector_View.TcIO
INTERFACE ITF_BaseGroupElement_HMI_Connector_View EXTENDS ITF_BaseControlElement_HMI_Connector_View

END_INTERFACE

// ---- POUs/A07_FB_BaseTopElement/ITF_BaseTopElement_HMI_Connector_View.TcIO
INTERFACE ITF_BaseTopElement_HMI_Connector_View EXTENDS ITF_BaseGroupElement_HMI_Connector_View

END_INTERFACE

// ---- POUs/B02_Recipes/ITF_BaseCreatingTemplateMethod.TcIO
(*			
	RafalOS
	Rafał Osajda		26.11.2025		TC 4024.66
	Wydzielone metody do tworzenia szablonu receptury
*)
INTERFACE ITF_BaseCreatingTemplateMethod

(*			
	RafalOS
	Rafał Osajda		25.10.2025		TC 4024.66
	Dodawanie składnika do szablonu
*)
METHOD PUBLIC AddIngredientToTemplate : BOOL
VAR_INPUT
	uiNumber		: UINT;
	stIngredient	: ST_BaseDescriptor;
END_VAR
END_METHOD

(*			
	RafalOS
	Rafał Osajda		25.10.2025		TC 4024.66
	Dodawanie szablonu - metoda wykorzystywana w zewnętrznym FB tworzenia receptur
*)
METHOD PUBLIC AddTemplate : BOOL
VAR_INPUT
	stTexts			: ST_BaseLabel;
END_VAR
END_METHOD

METHOD PUBLIC GetNumberIngredientOFTemplate : UINT
VAR_INPUT
	uiNumber				: UINT;
END_VAR
END_METHOD

METHOD PUBLIC GetNumberOfTemplate : UINT
VAR_INPUT
END_VAR
END_METHOD

END_INTERFACE

// ---- POUs/B02_Recipes/ITF_BaseRecipe.TcIO
(*			
	RafalOS
	Rafał Osajda		28.02.2025		TC 4026.13		wer. 0.0.0.1
	Obsługa receptur
*)
INTERFACE ITF_BaseRecipe

(*			
	RafalOS
	Rafał Osajda		25.10.2025		TC 4024.66
	Dodanie itferfejsu FB dla tworzenia szablonów receptur z programu maszyny
*)
METHOD PUBLIC AddITFToCreateTemplate : BOOL
VAR_INPUT
	fbToCtreateTemplate		: ITF_BaseCreateTemplateOfRecipe;
END_VAR
END_METHOD

(*			
	RafalOS
	Rafał Osajda		03.03.2025		TC 4026.13		wer. 0.0.0.1
	Kopiuje składniki z wybranej receptury i tworzy nową recepture
*)
METHOD PUBLIC AddRecipeFromRecipe : BOOL
VAR_INPUT
	uiNumberRecipe				: UINT;
	stTexts						: ST_BaseLabel;
END_VAR
END_METHOD

(*			
	RafalOS
	Rafał Osajda		03.03.2025		TC 4026.13		wer. 0.0.0.1
	Kopiuje składniki z wybranego szablonu i tworzy nową recepture
*)
METHOD PUBLIC AddRecipeFromTemplate : BOOL
VAR_INPUT
	uiNumberTemplates			: UINT;
	stTexts						: ST_BaseLabel;
END_VAR
END_METHOD

(*			
	RafalOS
	Rafał Osajda		03.03.2025		TC 4026.13		wer. 0.0.0.1
	Przypisuje do referencji wybraną rtecepture
*)
METHOD PUBLIC Choose : BOOL
VAR_INPUT
	uiNumber				: UINT;
END_VAR
END_METHOD

(*			
	RafalOS
	Rafał Osajda		03.06.2025		TC 4024.66
	usuwa referencje do wybranej
*)
METHOD PUBLIC ClearChosen
VAR_INPUT
END_VAR
END_METHOD

(*			
	RafalOS
	Rafał Osajda		25.10.2025		TC 4024.66
	Utworzenie nowych szablonów receptur na podstawie dodanych fb zewnętrznych - wywołanie metody powoduje
	skosowanie dotychczasowych szablonów i receptur
*)
METHOD PUBLIC CreateTemplates : BOOL
VAR_INPUT
END_VAR
END_METHOD

(*			
	RafalOS
	Rafał Osajda		03.03.2025		TC 4026.13		wer. 0.0.0.1
	
*)
METHOD PUBLIC DeleteRecipe : BOOL
VAR_INPUT
	uiNumber				: uint;
END_VAR
END_METHOD

(*			
	RafalOS
	Rafał Osajda		30.04.2025		TC 4024.66
	usunięcie wszystkich receptur
*)
METHOD PUBLIC DeleteRecipes : BOOL
VAR_INPUT
END_VAR
END_METHOD

(*			
	RafalOS
	Rafał Osajda		03.03.2025		TC 4026.13		wer. 0.0.0.1
	Zwraca referencje do  receptury
*)
METHOD PUBLIC GetChoosen : REFERENCE TO ST_BaseRecipe
END_METHOD

(*			
	RafalOS
	Rafał Osajda		03.03.2025		TC 4026.13		wer. 0.0.0.1
	
*)
METHOD PUBLIC GetIngredientFromRecipe : ST_BaseDescriptor
VAR_INPUT
	uiNumberOfRecipe			: UINT;
	uiNumberOfIngredient		: UINT;
END_VAR
END_METHOD

METHOD GetNamesOfRecipe : ST_BaseLabel
VAR_INPUT
	uiNumber			: UINT;
END_VAR
END_METHOD

METHOD PUBLIC GetNamesOfTemplate : ST_BaseLabel
VAR_INPUT
	uiNumber			: UINT;
END_VAR
END_METHOD

(*			
	RafalOS
	Rafał Osajda		03.03.2025		TC 4026.13		wer. 0.0.0.1
	
*)
METHOD PUBLIC GetNumberIngredientOfRecipe : UINT
VAR_INPUT
	uiNumber				: UINT;
END_VAR
END_METHOD

METHOD PUBLIC GetNumberIngredientOFTemplate : UINT
VAR_INPUT
	uiNumber				: UINT;
END_VAR
END_METHOD

METHOD PUBLIC GetNumberOfChoosen : UINT
VAR_INPUT
END_VAR
END_METHOD

METHOD PUBLIC GetNumberOfCreatingRecipe : UINT
VAR_INPUT
END_VAR
END_METHOD

METHOD PUBLIC GetNumberOfRecipe : UINT
VAR_INPUT
END_VAR
END_METHOD

METHOD PUBLIC GetNumberOfTemplate : UINT
VAR_INPUT
END_VAR
END_METHOD

(*			
	RafalOS
	Rafał Osajda		24.03.2025		TC 4024.66
	Zwraca reference do wybranej receptury
*)
METHOD PUBLIC GetReferencesToChoosen : REFERENCE TO ST_BaseRecipe
VAR_INPUT
END_VAR
END_METHOD

(*			
	RafalOS
	Rafał Osajda		03.03.2025		TC 4026.13		wer. 0.0.0.1
	Zwraca referencje do  receptury
*)
METHOD PUBLIC GetReferenceToRecipe : REFERENCE TO ST_BaseRecipe
VAR_INPUT
	uiNumer					: UINT;
END_VAR
END_METHOD

METHOD PUBLIC IsChoosen : BOOL
VAR_INPUT
END_VAR
END_METHOD

(*			
	RafalOS
	Rafał Osajda		03.03.2025		TC 4026.13		wer. 0.0.0.1
	Zastępuje wybraną recepture przez istenijącą receputre
*)
METHOD PUBLIC ReplaceRecipeWithAnotherRecipe : BOOL
VAR_INPUT
	uiNumerRecepturyCel			: UINT;
	uiNumerRecepturyZrodlo		: UINT;	
	stNazwa						: ST_BaseLabel;
END_VAR
END_METHOD

(*			
	RafalOS
	Rafał Osajda		03.03.2025		TC 4026.13		wer. 0.0.0.1
	Zastępuje wybraną recepture przez istenijącą receputre z szablonu
*)
METHOD PUBLIC ReplaceRecipeWithTemplateRecipe : BOOL
VAR_INPUT
	uiNumerRecepturyCel			: UINT;
	uiNumerRecepturyZrodlo		: UINT;
	stNazwa						: ST_BaseLabel;
END_VAR
END_METHOD

(*			
	RafalOS
	Rafał Osajda		05.12.2025		TC 4024.66
	Ustawia nową wartośc w podanym składniku
*)
METHOD PUBLIC SetIngredientValue
VAR_INPUT
	iRecipe			: int;
	iIngredient		: INT;
	rValue			: REAL;
END_VAR
END_METHOD

END_INTERFACE

// ---- POUs/B02_Recipes/ITF_BaseRecipe_HMI_Connector.TcIO
INTERFACE ITF_BaseRecipe_HMI_Connector

(*			
	RafalOS
	Rafał Osajda		03.03.2025		TC 4026.13		wer. 0.0.0.1
	Kopiuje składniki z wybranej receptury i tworzy nową recepture
*)
METHOD PUBLIC AddRecipeFromRecipe : BOOL
VAR_INPUT
	uiNumberRecipe				: UINT;
	stTexts						: ST_BaseLabel;
END_VAR
END_METHOD

(*			
	RafalOS
	Rafał Osajda		03.03.2025		TC 4026.13		wer. 0.0.0.1
	Kopiuje składniki z wybranego szablonu i tworzy nową recepture
*)
METHOD PUBLIC AddRecipeFromTemplate : BOOL
VAR_INPUT
	uiNumberTemplates			: UINT;
	stTexts						: ST_BaseLabel;
END_VAR
END_METHOD

(*			
	RafalOS
	Rafał Osajda		03.03.2025		TC 4026.13		wer. 0.0.0.1
	Przypisuje do referencji wybraną rtecepture
*)
METHOD PUBLIC Choose : BOOL
VAR_INPUT
	uiNumber				: UINT;
END_VAR
END_METHOD

(*			
	RafalOS
	Rafał Osajda		03.06.2025		TC 4024.66
	usuwa referencje do wybranej
*)
METHOD PUBLIC ClearChosen
VAR_INPUT
END_VAR
END_METHOD

(*			
	RafalOS
	Rafał Osajda		25.10.2025		TC 4024.66
	Utworzenie nowych szablonów receptur na podstawie dodanych fb zewnętrznych - wywołanie metody powoduje
	skosowanie dotychczasowych szablonów i receptur
*)
METHOD PUBLIC CreateTemplates : BOOL
VAR_INPUT
END_VAR
END_METHOD

(*			
	RafalOS
	Rafał Osajda		03.03.2025		TC 4026.13		wer. 0.0.0.1
	
*)
METHOD PUBLIC DeleteRecipe : BOOL
VAR_INPUT
	uiNumber				: uint;
END_VAR
END_METHOD

(*			
	RafalOS
	Rafał Osajda		03.03.2025		TC 4026.13		wer. 0.0.0.1
	
*)
METHOD PUBLIC GetIngredientFromRecipe : ST_BaseDescriptor
VAR_INPUT
	uiNumberOfRecipe			: UINT;
	uiNumberOfIngredient		: UINT;
END_VAR
END_METHOD

(*			
	RafalOS
	Rafał Osajda		02.12.2025		TC 4024.66
	Zwraca do tablicy wybrany zakres składników
*)
METHOD PUBLIC GetIngredientRange 
VAR_INPUT
	iRecipe			: INT;	//numer receptury z której bierzemy składniki
	iStartIndex		: INT;	//numer startowy składnika
	iCount			: INT;	//ilośc pobieranych 
END_VAR
VAR_IN_OUT
	arrOut : ARRAY [*] OF ST_BaseDescriptor;
END_VAR
VAR_OUTPUT
	iNumberOfFilledData	: INT;	//ilosc wypelnionych danych na strone
END_VAR
END_METHOD

METHOD GetNameList : ST_BaseRecipeList
VAR_INPUT
END_VAR
END_METHOD

METHOD GetNameListTemplate : ST_BaseRecipeList
END_METHOD

METHOD GetNamesOfSelectRecipe : ST_BaseLabel
VAR_INPUT

END_VAR
END_METHOD

(*			
	RafalOS
	Rafał Osajda		03.03.2025		TC 4026.13		wer. 0.0.0.1
	
*)
METHOD PUBLIC GetNumberIngredientOfRecipe : UINT
VAR_INPUT
	uiNumber				: UINT;
END_VAR
END_METHOD

METHOD PUBLIC GetNumberOfChoosen : UINT
VAR_INPUT
END_VAR
END_METHOD

METHOD PUBLIC GetNumberOfRecipe : UINT
VAR_INPUT
END_VAR
END_METHOD

METHOD PUBLIC GetNumberOfTemplate : UINT
VAR_INPUT
END_VAR
END_METHOD

METHOD PUBLIC IsChoosen : BOOL
VAR_INPUT
END_VAR
END_METHOD

(*			
	RafalOS
	Rafał Osajda		05.12.2025		TC 4024.66
	Ustawia nową wartośc w podanym składniku
*)
METHOD PUBLIC SetIngredientValue
VAR_INPUT
	iRecipe			: int;
	iIngredient		: INT;
	rValue			: REAL;
END_VAR
END_METHOD

END_INTERFACE

// ---- POUs Compilation/PRG_Compilation.TcPOU
PROGRAM PRG_Compilation
VAR
	fbLabel					: FB_BaseLabel;
	fbDescription			: FB_BaseDescriptor;
	fbLocation				: FB_BaseLocation;
	fbCommand				: FB_BaseCommand;
	fbImpuls				: FB_BaseImpulse;
	
	sttmpCommonData			: ST_BaseCommonData;

	fbBaseTime				: FB_BaseTime;
	fbBaseCommand			: FB_BaseCommand;
	fbBaseDescriptor		: FB_BaseDescriptor;
	fbBaseFlag				: FB_BaseFlag;
	fbBaseImplulse			: FB_BaseImpulse;
	fbBaseLocation			: FB_BaseLocation;
	
	fbBaseLogger			: FB_BaseLogger;
	fbBaseLoggerElement		: FB_BaseLoggerElement;
	fbBaseComponent			: FB_BaseComponent;
	fbBaseExecutiveElement	: FB_BaseControlElement;
	fbBaseComplexElement	: FB_BaseGroupElement;
	fbBaseMainComponent		: FB_BaseTopElement;
//B
	fbKomunikator		: FB_BaseCommunicator;
	fbReceptury			: FB_BaseRecipe;	
END_VAR

END_PROGRAM

// ---- POUs/A00_Basic/FB_BaseLabel.TcPOU
(*			
	RAFALOS
	Rafał Osajda		19.09.2025		TC 4024.66
	
*)
FUNCTION_BLOCK FB_BaseLabel IMPLEMENTS ITF_BaseLabel
VAR
	stTexts						: ST_BaseLabel;
END_VAR

METHOD PUBLIC GetTexts : ST_BaseLabel
VAR_INPUT
END_VAR
GetTexts				:=THIS^.stTexts;
END_METHOD

METHOD PUBLIC SetText
VAR_INPUT
	eLocation			: E_BaseLocation;
	wsDescription		: WSTRING;
END_VAR
THIS^.stTexts.arrText [eLocation]	:= wsDescription;
END_METHOD

METHOD PUBLIC SetTexts
VAR_INPUT
	stTexts				: ST_BaseLabel;
END_VAR
THIS^.stTexts			:= stTexts;
END_METHOD

END_FUNCTION_BLOCK

// ---- POUs/A00_Basic/FB_BaseDescriptor.TcPOU
(*			
	RAFALOS
	Rafał Osajda		19.09.2025		TC 4024.66
	
*)
FUNCTION_BLOCK FB_BaseDescriptor IMPLEMENTS ITF_BaseDescriptor
VAR
	stDescriptor					: ST_BaseDescriptor;
END_VAR

METHOD PUBLIC GetDefaultValue : REAL
VAR_INPUT
END_VAR
GetDefaultValue			:= THIS^.stDescriptor.rDefaultValue;
END_METHOD

METHOD PUBLIC GetDefaultValueFrom : REAL
VAR_INPUT
	stIN				: ST_BaseDescriptor;
END_VAR
GetDefaultValueFrom			:= stIN.rDefaultValue;
END_METHOD

METHOD PUBLIC GetDescriptor : ST_BaseDescriptor
VAR_INPUT
END_VAR
GetDescriptor		:= this^.stDescriptor;
END_METHOD

METHOD PUBLIC GetMax : REAL
VAR_INPUT
END_VAR
GetMax					:= THIS^.stDescriptor.rMax;
END_METHOD

METHOD PUBLIC GetMaxFrom : REAL
VAR_INPUT
	stIN				: ST_BaseDescriptor;
END_VAR
GetMaxFrom				:= stIN.rMax;
END_METHOD

METHOD PUBLIC GetMin : REAL
VAR_INPUT
END_VAR
GetMin				:= THIS^.stDescriptor.rMin;
END_METHOD

METHOD PUBLIC GetMinFrom : REAL
VAR_INPUT
	stIN			: ST_BaseDescriptor;
END_VAR
GetMinFrom			:= stIN.rMin;
END_METHOD

METHOD PUBLIC GetTexts : ST_BaseLabel
VAR_INPUT
END_VAR
GetTexts				:=THIS^.stDescriptor.stTexts;
END_METHOD

METHOD PUBLIC GetTextsFrom : ST_BaseLabel
VAR_INPUT
	stIN				: ST_BaseDescriptor;
END_VAR
GetTextsFrom			:=stIN.stTexts;
END_METHOD

METHOD PUBLIC GetUnit : STRING(6)
VAR_INPUT
END_VAR
GetUnit			:= THIS^.stDescriptor.sUnit;
END_METHOD

METHOD PUBLIC GetUnitFrom : STRING(6)
VAR_INPUT
	stIN			: ST_BaseDescriptor;
END_VAR
GetUnitFrom			:= stIN.sUnit;
END_METHOD

METHOD PUBLIC GetValue : REAL
VAR_INPUT
END_VAR
GetValue			:= this^.stDescriptor.rValue;
END_METHOD

METHOD PUBLIC GetValueFrom : REAL
VAR_INPUT
	stIN			: ST_BaseDescriptor;
END_VAR
GetValueFrom		:= stIN.rValue;
END_METHOD

METHOD PUBLIC SetDefaultValue
VAR_INPUT
	rDefaultValue: REAL;
END_VAR
THIS^.stDescriptor.rDefaultValue		:= rDefaultValue;
END_METHOD

METHOD PUBLIC SetDefaultValueIn
VAR_INPUT
	stIN			: REFERENCE TO ST_BaseDescriptor;
	rDefaultValue	: REAL;
END_VAR
stIN.rDefaultValue		:= rDefaultValue;
END_METHOD

METHOD PUBLIC SetMax
VAR_INPUT
	rMax: REAL;
END_VAR
THIS^.stDescriptor.rMax		:= rMax;
END_METHOD

METHOD PUBLIC SetMaxIn
VAR_INPUT
	stIN			: REFERENCE TO ST_BaseDescriptor;
	rMax: REAL;
END_VAR
stIN.rMax		:= rMax;
END_METHOD

METHOD PUBLIC SetMin
VAR_INPUT
	rMin: REAL;
END_VAR
THIS^.stDescriptor.rMin		:= rMin;
END_METHOD

METHOD PUBLIC SetMinIn
VAR_INPUT
	stIN			: REFERENCE TO ST_BaseDescriptor;
	rMin: REAL;
END_VAR
stIn.rMin		:= rMin;
END_METHOD

METHOD PUBLIC SetText
VAR_INPUT
	eLocation			: E_BaseLocation;
	wsDescription		: WSTRING;
END_VAR
THIS^.stDescriptor.stTexts.arrText [eLocation]	:= wsDescription;
END_METHOD

METHOD PUBLIC SetTextIn
VAR_INPUT
	stIN				: REFERENCE TO ST_BaseDescriptor;
	eLocation			: E_BaseLocation;
	wsDescription		: WSTRING;
END_VAR
stIN.stTexts.arrText [eLocation]	:= wsDescription;
END_METHOD

METHOD PUBLIC SetTexts
VAR_INPUT
	stTexts				: ST_BaseLabel;
END_VAR
THIS^.stDescriptor.stTexts			:= stTexts;
END_METHOD

METHOD PUBLIC SetTextsIn
VAR_INPUT
	stIN				: REFERENCE TO ST_BaseDescriptor;
	stTexts				: ST_BaseLabel;
END_VAR
stIN.stTexts			:= stTexts;
END_METHOD

METHOD PUBLIC SetUnit
VAR_INPUT
	sUnit: STRING(6);
END_VAR
THIS^.stDescriptor.sUnit		:= sUnit;
END_METHOD

METHOD PUBLIC SetUnitIn
VAR_INPUT
	stIN			: REFERENCE TO ST_BaseDescriptor;
	sUnit: STRING(6);
END_VAR
stIN.sUnit		:= sUnit;
END_METHOD

METHOD PUBLIC SetValue
VAR_INPUT
	rValue: REAL;
END_VAR
THIS^.stDescriptor.rValue		:= rValue;
END_METHOD

METHOD PUBLIC SetValueIn
VAR_INPUT
	stIN			: REFERENCE TO ST_BaseDescriptor;
	rValue			: REAL;
END_VAR
stIN.rValue			:= rValue;
END_METHOD

END_FUNCTION_BLOCK

// ---- POUs/A00_Basic/FB_BaseFlag.TcPOU
(*			
	RAFALOS
	Rafał Osajda		19.09.2025		TC 4024.66
	
*)
FUNCTION_BLOCK FB_BaseFlag IMPLEMENTS ITF_BaseFlag
VAR
	bState				: BOOL;
END_VAR

METHOD PUBLIC GetFlag : BOOL
VAR_INPUT
END_VAR
GetFlag			:= THIS^.bState;
END_METHOD

METHOD PUBLIC SetFlag
VAR_INPUT
	bState				: BOOL;
END_VAR
THIS^.bState			:= bState;
END_METHOD

END_FUNCTION_BLOCK

// ---- POUs/A03_FB_BaseLoggerElement/FB_BaseLoggerElement.TcPOU
(*			
	RAFALOS
	Rafał Osajda		19.09.2025		TC 4024.66
	Element bazowy umożliwiający potomkom wysyłaś zgłoszenia do logera
*)
FUNCTION_BLOCK FB_BaseLoggerElement EXTENDS FB_Base IMPLEMENTS ITF_BaseLoggerElement, 
		ITF_BaseLoggerElement_HMI_Connector, ITF_BaseLogger_Item, ITF_DecoratedElement
VAR
	stIdentifier					: ST_BaseElementIdentifier;	//Identyfikacja elementu
	stEvents						: ST_BaseEvents;			//dane elementu dotyczące zdarzeń
END_VAR

(*			
	RafalOS
	Rafał Osajda		24.03.2025		TC 4024.66
	Dodawanie zgłoszenia do systemu
*)
METHOD PUBLIC AddEvent : BOOL
VAR_INPUT
	bIgnoreRepetitions					: BOOL;						//jak true nie zliczaj powtorzeń wystapienia np komunikaty
	eEventCategory						: E_BaseEvents_Category;	//BYTE;	//1 - blad, 2 - ostrzezenie, 3 - wiadomosc, 4 - safety
	bConfirm							: BOOL;						//wymaga powtierdzenia
	stDescription						: ST_BaseLabel;
END_VAR
IF (THIS^.stEvents.uiNumberOfAdded + 1 <= GVL_BaseConstans.MAX_EVENTS_PER_ITEM) THEN
	THIS^.stEvents.uiNumberOfAdded														:= THIS^.stEvents.uiNumberOfAdded + 1;
	THIS^.stEvents.arrDefinitions [THIS^.stEvents.uiNumberOfAdded].uiIDInItem			:= THIS^.stEvents.uiNumberOfAdded;
	THIS^.stEvents.arrDefinitions [THIS^.stEvents.uiNumberOfAdded].bIgnoreRepetitions	:= bIgnoreRepetitions;
	THIS^.stEvents.arrDefinitions [THIS^.stEvents.uiNumberOfAdded].eEventCategory		:= eEventCategory;
	THIS^.stEvents.arrDefinitions [THIS^.stEvents.uiNumberOfAdded].stDescription		:= stDescription;
	THIS^.stEvents.arrDefinitions [THIS^.stEvents.uiNumberOfAdded].bConfirm				:= bConfirm;
	AddEvent						:= TRUE;
ELSE
	AddEvent						:= FALSE;
END_IF
END_METHOD

METHOD PROTECTED EventAcknowledge : BOOL
VAR_INPUT
	iNumber				: INT;
END_VAR
VAR
	sttmpRow			: ST_BaseEvents_RowInQueue;
	btmpExit			: BOOL;
END_VAR
IF (iNumber > 0 AND iNumber <= TO_INT (THIS^.stEvents.uiNumberOfAdded)) THEN
	IF ((THIS^.stEvents.arrDefinitions [iNumber].bConfirm AND NOT THIS^.stEvents.arrConfirmation [iNumber]) OR NOT THIS^.stEvents.arrDefinitions [iNumber].bConfirm) THEN
		THIS^.stEvents.arrConfirmation [iNumber] 	:= TRUE;
		btmpExit									:= TRUE;
		IF (THIS^.stEvents.bLoggerDataCompleted) THEN
			sttmpRow.eEventAction		:= E_BaseEvents_Action.Confirm;
			sttmpRow.uiIDEvent			:= THIS^.stEvents.arrDefinitions [iNumber].uiIDEvent;
			sttmpRow.dtConfirmed		:= THIS^.refstCommonData.itfTime.StampDT ();
		
			THIS^.refstCommonData.itfLogger.ReportEvent (stEvent	:= sttmpRow);	
			btmpExit						:= btmpExit;
		ELSE
			btmpExit						:= FALSE;
		END_IF
	END_IF	
END_IF
EventAcknowledge					:= btmpExit;
END_METHOD

(*			
	RafalOS
	Rafał Osajda		09.06.2025		TC 4024.66
	Szuka czy ma zgłoszenie i zadanym ID jak tak to usuwa i zwraca true w przeciwnym razie zwraca false 
*)
METHOD PUBLIC EventAcknowledgeByID : BOOL
VAR_INPUT
	uiIDEvent				: UINT;
END_VAR

VAR
	iI: INT;
	bResult: BOOL;
END_VAR
FOR iI := 1 TO TO_INT (THIS^.stEvents.uiNumberOfAdded) DO
	IF (THIS^.stEvents.arrDefinitions [iI].uiIDEvent = uiIDEvent AND THIS^.stEvents.arrDefinitions [iI].bConfirm) THEN	//Zgłoszenie znalezione
		IF (THIS^.EventAcknowledge (iNumber	:= iI)) THEN
			bResult							:= TRUE;
			EXIT;
		END_IF
	END_IF
END_FOR
EventAcknowledgeByID					:= bResult;
END_METHOD

METHOD PROTECTED EventDoesRequireConfirmation : BOOL
VAR_INPUT
	iNumber				: INT;
END_VAR
EventDoesRequireConfirmation		:= THIS^.stEvents.arrDefinitions [iNumber].bConfirm;
END_METHOD

(*			RafalOS
	Rafał Osajda		16.10.2024		TC 4026.11		wer. 0.0.0.1
	Zwraca aktualny stan wybranego zgłoszenia
*)
METHOD PROTECTED EventIsActive : BOOL
VAR_INPUT
	iNumber					: INT;
END_VAR
IF (iNumber > 0 AND iNumber <= TO_INT (THIS^.stEvents.uiNumberOfAdded)) THEN
	EventIsActive			:= THIS^.stEvents.arrState [iNumber];
END_IF
END_METHOD

(*			
	RafalOS
	Rafał Osajda		24.03.2025		TC 4024.66
	Definicja nowego zgłoszenia
*)
METHOD PUBLIC EventsDefinition : BOOL
MEMSET (
	destAddr		:= ADR (THIS^.stEvents.arrDefinitions),
	fillByte		:= 0,
	n				:= SIZEOF (THIS^.stEvents.arrDefinitions)
);
THIS^.stEvents.uiNumberOfAdded	:= 0;
END_METHOD

(*			
	RafalOS
	Rafał Osajda		24.03.2025		TC 4024.66
	Zgloszenie nowe wlacz 
*)
METHOD PROTECTED EventSetActive : BOOL
VAR_INPUT
	iNumber					: INT; //numer zgloszenia w elemencie
END_VAR
VAR
	sttmpRow				: ST_BaseEvents_RowInQueue;
END_VAR
IF (iNumber > 0 AND iNumber <= TO_INT (THIS^.stEvents.uiNumberOfAdded) AND NOT THIS^.stEvents.arrState [iNumber]) THEN
	THIS^.stEvents.arrState [iNumber]		:= TRUE;
	IF (NOT THIS^.stEvents.arrDefinitions [iNumber].bIgnoreRepetitions) THEN
		THIS^.stEvents.arrDefinitions [iNumber].uiRepetitionCounter := THIS^.stEvents.arrDefinitions [iNumber].uiRepetitionCounter + 1;
	END_IF
	IF (THIS^.stEvents.bLoggerDataCompleted) THEN
		sttmpRow.eEventAction		:= E_BaseEvents_Action.Start;
		sttmpRow.uiIDEvent			:= THIS^.stEvents.arrDefinitions [iNumber].uiIDEvent;
		sttmpRow.bActive			:= TRUE;
		sttmpRow.bIgnoreRepetitions	:= THIS^.stEvents.arrDefinitions [iNumber].bIgnoreRepetitions;
		sttmpRow.dtStart			:= THIS^.refstCommonData.itfTime.StampDT ();
		sttmpRow.uiRepetitionCounter:= THIS^.stEvents.arrDefinitions [iNumber].uiRepetitionCounter;
		sttmpRow.eEventCategory		:= THIS^.stEvents.arrDefinitions [iNumber].eEventCategory;
		sttmpRow.bConfirm			:= THIS^.stEvents.arrDefinitions [iNumber].bConfirm;
		sttmpRow.uiIDItem			:= THIS^.stIdentifier.uiID;
		
		THIS^.refstCommonData.itfLogger.ReportEvent (stEvent := sttmpRow);
		THIS^.stEvents.iNumberOfActiveEvents	:= THIS^.stEvents.iNumberOfActiveEvents + 1;
	END_IF
END_IF
END_METHOD

(*			
	RafalOS
	Rafał Osajda		24.03.2025		TC 4024.66
	Zgloszenie zakonczone wylacz
*)
METHOD PROTECTED EventSetInactive : BOOL
VAR_INPUT
	iNumber				: INT;
END_VAR
VAR
	iI					: INT;
	sttmpRow			: ST_BaseEvents_RowInQueue;
	btmpExit			: BOOL := FALSE;
END_VAR
IF (iNumber > 0 AND iNumber <= TO_INT (THIS^.stEvents.uiNumberOfAdded) AND THIS^.stEvents.arrState [iNumber]) THEN
	IF ((THIS^.stEvents.arrDefinitions [iNumber].bConfirm AND THIS^.stEvents.arrConfirmation [iNumber]) OR NOT THIS^.stEvents.arrDefinitions [iNumber].bConfirm) THEN
		stEvents.arrState [iNumber]					:= FALSE;
		THIS^.stEvents.arrConfirmation [iNumber]	:= FALSE;
		btmpExit									:= TRUE;
	END_IF
	IF (THIS^.stEvents.bLoggerDataCompleted) THEN
		sttmpRow.eEventAction		:= E_BaseEvents_Action.Stop;
		sttmpRow.uiIDEvent			:= THIS^.stEvents.arrDefinitions [iNumber].uiIDEvent;
		sttmpRow.dtFinish			:= THIS^.refstCommonData.itfTime.StampDT ();
		sttmpRow.bActive			:= FALSE;
	
		THIS^.refstCommonData.itfLogger.ReportEvent (stEvent	:= sttmpRow);
		THIS^.stEvents.iNumberOfActiveEvents	:= THIS^.stEvents.iNumberOfActiveEvents - 1;
		btmpExit						:= btmpExit;
	ELSE
		btmpExit						:= FALSE;
	END_IF
END_IF
EventSetInactive 						:= btmpExit;
END_METHOD

(*			
	RafalOS
	Rafał Osajda		09.06.2025		TC 4024.66
	Szuka czy ma zgłoszenie i zadanym ID jak tak to usuwa i zwraca true w przeciwnym razie zwraca false 
*)
METHOD PUBLIC EventSetInactiveByID : BOOL
VAR_INPUT
	uiIDEvent				: UINT;
END_VAR

VAR
	iI: INT;
	bResult: BOOL;
END_VAR
FOR iI := 1 TO TO_INT (THIS^.stEvents.uiNumberOfAdded) DO
	IF (THIS^.stEvents.arrDefinitions [iI].uiIDEvent = uiIDEvent AND
		((NOT THIS^.stEvents.arrDefinitions [iI].bConfirm) OR 
			(THIS^.stEvents.arrDefinitions [iI].bConfirm AND THIS^.stEvents.arrConfirmation [iI]))) THEN	//Zgłoszenie znalezione
		IF (THIS^.EventSetInactive (iNumber := iI)) THEN
			bResult							:= TRUE;
			EXIT;
		END_IF
	END_IF
END_FOR
EventSetInactiveByID						:= bResult;
END_METHOD

(*			
	RAFALOS
	Rafał Osajda		25.09.2025		TC 4024.66
	Metoda wywoływana w pierwszym cyklu
*)
METHOD PUBLIC FirstCycle : BOOL
VAR_INPUT
END_VAR
	(*	Zdefiniowanie zdarzeń dla elementu	*)
THIS^.EventsDefinition ();


FirstCycle					:= TRUE;
END_METHOD

METHOD PUBLIC GetCode : STRING
VAR_INPUT
END_VAR
GetCode			:= THIS^.stIdentifier.sCode;
END_METHOD

METHOD PUBLIC GetID : UINT
VAR_INPUT
END_VAR
GetID				:= THIS^.stIdentifier.uiID;
END_METHOD

METHOD PUBLIC GetIdentyfier : ST_BaseElementIdentifier
VAR_INPUT
END_VAR
GetIdentyfier				:= THIS^.stIdentifier;
END_METHOD

METHOD GetInformationToDisplayEvent : ST_BaseLogger_ItemDataToDisplay
VAR_INPUT
	uiIDEvent				: UINT;
END_VAR
VAR
	sttmpResult				: ST_BaseLogger_ItemDataToDisplay;
	iI: INT;
END_VAR
sttmpResult.stItemName		:= THIS^.stIdentifier.stName;
sttmpResult.sCode			:= THIS^.stIdentifier.sCode;
FOR iI := 1 TO TO_INT (THIS^.stEvents.uiNumberOfAdded) DO 
	IF (THIS^.stEvents.arrDefinitions [iI].uiIDEvent = uiIDEvent) THEN
		sttmpResult.stDescription	:= THIS^.stEvents.arrDefinitions [iI].stDescription;
		sttmpResult.eEventCategory	:= THIS^.stEvents.arrDefinitions [iI].eEventCategory;
		sttmpResult.sEventCategory	:= TO_STRING (THIS^.stEvents.arrDefinitions [iI].eEventCategory);
		sttmpResult.uiRepetitionCounter	:= THIS^.stEvents.arrDefinitions [iI].uiRepetitionCounter;
		EXIT;
	END_IF
END_FOR

GetInformationToDisplayEvent	:= sttmpResult;
END_METHOD

METHOD GetITFComponent : ITF_BaseComponent
VAR_INPUT
END_VAR
GetITFComponent		:= null;
END_METHOD

METHOD GetITFControlElement : ITF_BaseControlElement
VAR_INPUT
END_VAR
GetITFControlElement	:= null;
END_METHOD

METHOD GetITFGroupElement : ITF_BaseGroupElement
VAR_INPUT
END_VAR
GetITFGroupElement	:= null;
END_METHOD

METHOD GetITFLoggerElement : ITF_BaseLoggerElement
VAR_INPUT
END_VAR
GetITFLoggerElement		:= THIS^;
END_METHOD

METHOD GetITFTopElement : ITF_BaseTopElement
VAR_INPUT
END_VAR
GetITFTopElement		:= null;
END_METHOD

METHOD PUBLIC GetName : ST_BaseLabel
VAR_INPUT
END_VAR
GetName				:= THIS^.stIdentifier.stName;
END_METHOD

METHOD PUBLIC GetType : E_BaseElementType
VAR_INPUT
END_VAR
GetType				:= THIS^.stIdentifier.eType;
END_METHOD

METHOD PUBLIC LinkCommonData : BOOL
VAR_INPUT
	stCommonData				: REFERENCE TO ST_BaseCommonData;
END_VAR
VAR
	bResult						: BOOL;
END_VAR
bResult		:= SUPER^.LinkCommonData (stCommonData := stCommonData);

(* sprawdzenie czy jest podłaczony loger	*)
THIS^.stEvents.bLoggerDataCompleted	:= THIS^.refstCommonData.itfLogger <> 0;

LinkCommonData		:= bResult AND THIS^.stEvents.bLoggerDataCompleted;
END_METHOD

METHOD PUBLIC SetCode
VAR_INPUT
	sCode							: STRING;
	sAdd							: STRING;
END_VAR
THIS^.stIdentifier.sCode				:= sCode;
END_METHOD

(*			
	RafalOS
	Rafał Osajda		03.10.2025		TC 4024.66
	nadawanie unikalnych ID dla zdarzeń
*)
METHOD PUBLIC SetEventsIDs : UINT
VAR_INPUT
	uiNewID		: UINT;
END_VAR
VAR
	uiI			: UINT;
	uitmpValue	: UINT;
	uitmpValue2	: UINT;
END_VAR
IF (THIS^.stEvents.uiNumberOfAdded > 0) THEN
	FOR uiI := 1 TO THIS^.stEvents.uiNumberOfAdded DO
		uitmpValue	:= SEL (uiNewID = 0, uiNewID, 1);
		uitmpValue2	:= uitmpValue + uiI;// - 1;
		THIS^.stEvents.arrDefinitions [uiI].uiIDEvent	:= uitmpValue2;
	END_FOR
	SetEventsIDs				:= uiNewID + THIS^.stEvents.uiNumberOfAdded;
ELSE
	SetEventsIDs				:= uiNewID;
END_IF
END_METHOD

METHOD PUBLIC SetID : UINT
VAR_INPUT
	uiID					: UINT;
END_VAR
THIS^.stIdentifier.uiID			:= uiID;
SetID							:= uiID;
END_METHOD

METHOD PUBLIC SetName
VAR_INPUT
	stName				: ST_BaseLabel;
END_VAR
this^.stIdentifier.stName			:= stName;
END_METHOD

METHOD PUBLIC SetType
VAR_INPUT
	eType					: E_BaseElementType;
END_VAR
THIS^.stIdentifier.eType				:= eType;
END_METHOD

METHOD PUBLIC ZwrocDaneDlaZgloszeniaOID : BOOL
VAR_INPUT
	uiIDZgloszenia				: UINT;
END_VAR
VAR_OUTPUT
	uiIDElementu				: UINT;
	sKodElementu				: STRING;
	sRodzajZgloszenia			: STRING;
	eRodzajZgloszenia			: E_BaseEvents_Category;
	stOpis						: ST_BaseLabel;
	stTekstElementu				: ST_BaseLabel;
END_VAR
VAR
	iI: INT;
END_VAR
FOR iI := 1 TO TO_INT (THIS^.stEvents.uiNumberOfAdded) DO
	IF (THIS^.stEvents.arrDefinitions [iI].uiIDEvent = uiIDElementu) THEN
		uiIDElementu				:= THIS^.stIdentifier.uiID;
	    sKodElementu				:= THIS^.stIdentifier.sCode;
	    sRodzajZgloszenia			:= TO_STRING (THIS^.stEvents.arrDefinitions [iI].eEventCategory);
	    eRodzajZgloszenia			:= THIS^.stEvents.arrDefinitions [iI].eEventCategory;
	    stOpis						:= THIS^.stEvents.arrDefinitions [iI].stDescription;
		stTekstElementu				:= THIS^.stIdentifier.stName;
		ZwrocDaneDlaZgloszeniaOID	:= TRUE;
		EXIT;
	END_IF
END_FOR
END_METHOD

END_FUNCTION_BLOCK

// ---- POUs/A04_FB_BaseComponent/FB_BaseComponent.TcPOU
(*			
	RAFALOS
	Rafał Osajda		19.09.2025		TC 4024.66
	Komponent bazowy dla elementów prostych
*)
FUNCTION_BLOCK FB_BaseComponent EXTENDS FB_BaseLoggerElement IMPLEMENTS ITF_BaseComponent, ITF_BaseComponent_HMI_Connector
VAR
	cmdReset						: FB_BaseCommand;
	cmdParametersCreate				: FB_BaseCommand;
	cmdParametersRestoreToDefault	: FB_BaseCommand;
	
	
END_VAR
VAR PERSISTENT
	stParameters					: ST_Parameters;
END_VAR

(*			
	RafalOS
	Rafał Osajda		27.03.2025		TC 4024.66
	Obsluga bledow sprawdzanie czy jakis blad sie nei pojawil i ustawienie stanu lub wylaczenie
*)
METHOD PUBLIC ExecuteEveryCycle_Error
VAR_INPUT
END_VAR
END_METHOD

(*			
	RafalOS
	Rafał Osajda		27.03.2025		TC 4024.66
	Wywolanie co cykl operacji 
*)
METHOD PUBLIC ExecuteEveryCycle_Operation
VAR_INPUT
END_VAR
IF (THIS^.cmdReset.OperationExecute ()) THEN
	THIS^.cmdReset.Operation (bIN		:= THIS^.ResetOperation ());
END_IF

IF (THIS^.cmdParametersCreate.OperationExecute ()) THEN
	THIS^.cmdParametersCreate.Operation (bIN := THIS^.ParameterCreateTable ());
END_IF

IF (THIS^.cmdParametersRestoreToDefault.OperationExecute ()) THEN
	THIS^.cmdParametersRestoreToDefault.Operation (bIN	:= THIS^.ParameterRestoreDefaultValueAll ());
END_IF
END_METHOD

(*			
	RafalOS
	Rafał Osajda		27.03.2025		TC 4024.66
	Aktualizacja flag 
*)
METHOD PUBLIC ExecuteEveryCycle_Status
VAR_INST
END_VAR
END_METHOD

(*			
	RafalOS
	Rafał Osajda		27.03.2025		TC 4024.66
	Testowanie czy nei pojawil sie jakis rozkaz i uruchomienie odpowiednich operacji
*)
METHOD PUBLIC ExecuteEveryCycle_Test
VAR_INPUT
END_VAR
THIS^.cmdReset.Test ();
THIS^.cmdParametersCreate.Test ();
THIS^.cmdParametersRestoreToDefault.Test ();
END_METHOD

METHOD FB_init : BOOL
VAR_INPUT
	bInitRetains : BOOL; // if TRUE, the retain variables are initialized (warm start / cold start)
	bInCopyCode : BOOL;  // if TRUE, the instance afterwards gets moved into the copy code (online change)
END_VAR
THIS^.stIdentifier.eType			:= E_BaseElementType.eComponent;
END_METHOD

(*			
	RafalOS
	Rafał Osajda		03.10.2025		TC 4024.66
	
*)
METHOD PUBLIC FirstCycle : BOOL
VAR_INPUT
END_VAR
FirstCycle				:= SUPER^.FirstCycle ();
END_METHOD

METHOD GetITFComponent : ITF_BaseComponent
VAR_INPUT
END_VAR
GetITFComponent		:= THIS^;
END_METHOD

METHOD GetITFControlElement : ITF_BaseControlElement
VAR_INPUT
END_VAR
GetITFControlElement	:= null;
END_METHOD

METHOD GetITFGroupElement : ITF_BaseGroupElement
VAR_INPUT
END_VAR
GetITFGroupElement	:= null;
END_METHOD

METHOD GetITFTopElement : ITF_BaseTopElement
VAR_INPUT
END_VAR
GetITFTopElement		:= null;
END_METHOD

(*			
	RafalOS
	Rafał Osajda		07.10.2025		TC 4024.66
	Dodpisywanie się do listy logera
*)
METHOD PUBLIC JoinTheLogger : BOOL
VAR_INPUT
END_VAR
IF (THIS^.bIsValidCommonData) THEN
	IF (THIS^.refstCommonData.itfLogger.AddItem (itfItem := THIS^) > 0 ) THEN
		JoinTheLogger		:= TRUE;
	END_IF
END_IF
END_METHOD

(*			
	RafalOS
	Rafał Osajda		26.03.2025		TC 4024.66
	Dodawanie parametru do elementu wykonawczego - metode wywołać przy pierwszym uruchomieniu programu by wgrać parametry do pamięci
	później używać tylko edycji lub przywracania wartości domyślnych
*)
METHOD PUBLIC ParameterAdd : BOOL
VAR_INPUT
	stParameter			: ST_BaseDescriptor;
END_VAR
IF (THIS^.stParameters.uiNumber + 1 <= TO_UINT (GVL_BaseConstans.MAX_NUMBER_OF_PARAMETERS)) THEN
	THIS^.stParameters.uiNumber 		:= THIS^.stParameters.uiNumber + 1;
	THIS^.stParameters.arrRow [THIS^.stParameters.uiNumber] 	:= stParameter;
	ParameterAdd				:= TRUE;
ELSE
	ParameterAdd				:= FALSE;
END_IF
END_METHOD

(*			
	RafalOS
	Rafał Osajda		26.03.2025		TC 4024.66
	Modyfikuje wartość domyślną w istniejącym parametrze - true jak się zmiana udała
*)
METHOD PUBLIC ParameterCorrectDefaultValue : BOOL
VAR_INPUT
	uiNumber			: UINT;
	rValue				: REAL;
END_VAR
IF (uiNumber > 0 AND uiNumber <= THIS^.stParameters.uiNumber) THEN
	IF (rValue >= THIS^.GetMinFrom (stIN := THIS^.stParameters.arrRow [uiNumber]) AND
		rValue <= THIS^.GetMaxFrom (stIN := THIS^.stParameters.arrRow [uiNumber])) THEN
		THIS^.SetDefaultValueIn (stIN := THIS^.stParameters.arrRow [uiNumber], rDefaultValue	:= rValue);
		ParameterCorrectDefaultValue		:= TRUE;
	ELSE
		ParameterCorrectDefaultValue		:= FALSE;
	END_IF
ELSE
	ParameterCorrectDefaultValue		:= FALSE;
END_IF
END_METHOD

METHOD PUBLIC ParameterCorrectName : BOOL
VAR_INPUT
	eLocation					: E_BaseLocation;
	uiNumberOfParameter			: UINT;
	wsDescription				: WSTRING;
END_VAR
THIS^.SetTextIn (
	stIN 			:= THIS^.stParameters.arrRow [uiNumberOfParameter],
	eLocation		:= eLocation,
	wsDescription	:= wsDescription
);
END_METHOD

(*			
	RafalOS
	Rafał Osajda		26.03.2025		TC 4024.66
	Modyfikuje wartość w istniejącym parametrze - true jak się zmiana udała
*)
METHOD PUBLIC ParameterCorrectValue : BOOL
VAR_INPUT
	uiNumber			: UINT;
	rValue				: REAL;
END_VAR
IF (uiNumber > 0 AND uiNumber <= THIS^.stParameters.uiNumber) THEN
	IF (rValue <= THIS^.GetMaxFrom (stIN := THIS^.stParameters.arrRow [uiNumber]) AND
		rValue >= THIS^.GetMinFrom (stIN := THIS^.stParameters.arrRow [uiNumber]) ) THEN
		THIS^.SetValueIn (
			stIN		:= THIS^.stParameters.arrRow [uiNumber],
			rValue		:= rValue
		);
		ParameterCorrectValue		:= TRUE;
	ELSE
		ParameterCorrectValue		:= FALSE;
	END_IF
ELSE
	ParameterCorrectValue		:= FALSE;
END_IF
END_METHOD

(*			
	RafalOS
	Rafał Osajda		31.03.2025		TC 4024.66
	Metoda wymazująca dotychczasowe dane z tablicy parametrów i przypisująca je od nowa
*)
METHOD PROTECTED ParameterCreateTable : BOOL
VAR_INPUT
END_VAR
MEMSET (
	destAddr			:= ADR (THIS^.stParameters.arrRow),
	fillByte			:= 0,
	n					:= SIZEOF (THIS^.stParameters.arrRow)
);
THIS^.stParameters.uiNumber	:= 0;

ParameterCreateTable := TRUE;
END_METHOD

METHOD PUBLIC ParameterGet : ST_BaseDescriptor
VAR_INPUT
	uiNumer				: UINT;
END_VAR
ParameterGet			:= THIS^.stParameters.arrRow [uiNumer];
END_METHOD

(*			
	RafalOS
	Rafał Osajda		26.03.2025		TC 4024.66
	Zwraca wartosc domyslna
*)
METHOD PUBLIC ParameterGetDefaultValue : REAL
VAR_INPUT
	uiNumber				: UINT;
END_VAR
IF (uiNumber > 0 AND uiNumber <= THIS^.stParameters.uiNumber) THEN
	ParameterGetDefaultValue			:= THIS^.GetDefaultValueFrom (stIN :=  THIS^.stParameters.arrRow [uiNumber]);
ELSE
	ParameterGetDefaultValue			:= 0;
END_IF
END_METHOD

(*			
	RafalOS
	Rafał Osajda		26.03.2025		TC 4024.66
	Zwraca wartość MAX
*)
METHOD PUBLIC ParameterGetMax : REAL
VAR_INPUT
	uiNumber				: UINT;
END_VAR
IF (uiNumber > 0 AND uiNumber <= THIS^.stParameters.uiNumber) THEN
	ParameterGetMax			:= THIS^.GetMaxFrom (stIN :=  THIS^.stParameters.arrRow [uiNumber]);
ELSE
	ParameterGetMax			:= 0;
END_IF
END_METHOD

(*			
	RafalOS
	Rafał Osajda		26.03.2025		TC 4024.66
	Zwraca wartość MIN
*)
METHOD PUBLIC ParameterGetMin : REAL
VAR_INPUT
	uiNumber				: UINT;
END_VAR
IF (uiNumber >= 0 AND uiNumber <= THIS^.stParameters.uiNumber) THEN
	ParameterGetMin			:= THIS^.GetMinFrom (stIN := THIS^.stParameters.arrRow [uiNumber]);
ELSE
	ParameterGetMin			:= 0;
END_IF
END_METHOD

METHOD PUBLIC ParameterGetNumberOfAdded : UINT
VAR_INPUT
END_VAR
ParameterGetNumberOfAdded			:= THIS^.stParameters.uiNumber;
END_METHOD

(*			
	RafalOS
	Rafał Osajda		26.03.2025		TC 4024.66
	Zwraca jednostke
*)
METHOD PUBLIC ParameterGetUnit : STRING(6)
VAR_INPUT
	uiNumber				: uINT;
END_VAR
IF (uiNumber > 0 AND uiNumber <= THIS^.stParameters.uiNumber) THEN
	ParameterGetUnit			:= THIS^.GetUnitFrom (stIN :=  THIS^.stParameters.arrRow [uiNumber]);
ELSE
	ParameterGetUnit			:= '';
END_IF
END_METHOD

(*			
	RafalOS
	Rafał Osajda		26.03.2025		TC 4024.66
	Zwraca wartość
*)
METHOD PUBLIC ParameterGetValue : REAL
VAR_INPUT
	uiNumber				: UINT;
END_VAR
IF (uiNumber > 0 AND uiNumber <= THIS^.stParameters.uiNumber) THEN
	ParameterGetValue			:= THIS^.GetValueFrom (stIN := THIS^.stParameters.arrRow [uiNumber]);
ELSE
	ParameterGetValue			:= 0;
END_IF
END_METHOD

(*			
	RafalOS
	Rafał Osajda		26.03.2025		TC 4024.66
	Modyfikacja istniejącego parametra jako przypisanie nowego deskryptora
*)
METHOD PUBLIC ParameterModify : BOOL
VAR_INPUT
	uiNumber			: UINT;
	stParameter			: ST_BaseDescriptor;
END_VAR
IF (uiNumber > 0 AND uiNumber <= THIS^.stParameters.uiNumber) THEN
	THIS^.stParameters.arrRow [uiNumber]	:= 	stParameter;
	ParameterModify		:= TRUE;
ELSE
	ParameterModify		:= FALSE;
END_IF
END_METHOD

METHOD PUBLIC ParameterRestoreDefaultValue : BOOL
VAR_INPUT
	uiNumber		: UINT;
END_VAR
IF (uiNumber > 0 AND uiNumber <= THIS^.stParameters.uiNumber) THEN
	THIS^.SetValueIn (stIN := THIS^.stParameters.arrRow [uiNumber], rValue := THIS^.GetDefaultValueFrom (stIN := THIS^.stParameters.arrRow [uiNumber]));
	ParameterRestoreDefaultValue	:= TRUE;
ELSE
	ParameterRestoreDefaultValue	:= FALSE;
END_IF
END_METHOD

METHOD PROTECTED ParameterRestoreDefaultValueAll : BOOL
VAR_INPUT
END_VAR

VAR
	iI					: INT;
	bResult				: bool;
END_VAR
bResult					:= TRUE;
FOR iI := 1 TO TO_INT (THIS^.stParameters.uiNumber) DO 
	bResult				:= bResult AND THIS^.ParameterRestoreDefaultValue (uiNumber := TO_UINT (iI));
END_FOR
END_METHOD

(*			
	RafalOS
	Rafał Osajda		04.05.2025		TC 4024.66
	Skasowanie i utworzenie tablicy parametrów od nowa 
*)
METHOD PUBLIC ParametersCreate : BOOL
THIS^.cmdParametersCreate.Execute ();
END_METHOD

(*			
	RafalOS
	Rafał Osajda		04.05.2025		TC 4024.66
	Przywrocenie parametrow - in na false to tylko ten element true razem z podelementami
*)
METHOD PUBLIC ParameterSetToDefault : BOOL
THIS^.cmdParametersRestoreToDefault.Execute ();
END_METHOD

METHOD PUBLIC Reset : BOOL
VAR_INPUT
END_VAR
THIS^.cmdReset.Execute ();
END_METHOD

METHOD PUBLIC ResetGetBusy : BOOL
VAR_INPUT
END_VAR
ResetGetBusy		:= THIS^.cmdReset.IsBusy ();
END_METHOD

METHOD PUBLIC ResetGetStatus : BOOL
VAR_INPUT
END_VAR
ResetGetStatus			:= THIS^.cmdReset.IsStatus ();
END_METHOD

METHOD PROTECTED ResetOperation : BOOL
VAR_INPUT
END_VAR


ResetOperation			:= FALSE;
END_METHOD

END_FUNCTION_BLOCK

// ---- POUs/A05_FB_BaseControlElement/FB_BaseControlElement.TcPOU
(*			
	RAFALOS
	Rafał Osajda		19.09.2025		TC 4024.66
	Rodzic dla wszystkich elementów wykonawczych
*)
FUNCTION_BLOCK FB_BaseControlElement EXTENDS FB_BaseComponent IMPLEMENTS ITF_BaseControlElement, ITF_BaseControlElement_HMI_Connector
VAR
	arrComponent			: ARRAY  [1..GVL_BaseConstans.MAX_ITEM_PER_ELEMENT] OF ITF_BaseComponent;
	uiNumberOfComponents	: UINT;
(*	Zasilanie	*)
	itfSS1					: ITF_BaseFlagGet;
	itfSTO					: ITF_BaseFlagGet;
	stPower					: ST_BaseControlElement_Power;
(*	Bazowanie	*)
	stHoming				: ST_BaseControlElement_Homing;
(*	Flagi główne elementów	*)
	bPosition0				: BOOL := TRUE;	//jak nie potrzebna to zostawić na true w przeciwnym przypadku przypisać odpowiednią logikę
	bDoNothing				: BOOL := TRUE;	//jak nie potrzebna to zostawić na true w przeciwnym przypadku przypisać odpowiednią logikę
	
END_VAR

METHOD PROTECTED AddComponent : BOOL
VAR_INPUT
	itfComponent				: ITF_BaseComponent;
END_VAR
IF (THIS^.uiNumberOfComponents + 1 <= GVL_BaseConstans.MAX_ITEM_PER_ELEMENT) THEN
	THIS^.uiNumberOfComponents		:= THIS^.uiNumberOfComponents + 1;
	THIS^.arrComponent [THIS^.uiNumberOfComponents]	:= itfComponent;
	AddComponent				:= TRUE;
ELSE
	;//zwrocenie zbyt dużo komponentow
END_IF
END_METHOD

(*			
	RafalOS
	Rafał Osajda		24.03.2025		TC 4024.66
	Definicja nowego zgłoszenia
*)
METHOD PUBLIC EventsDefinition : BOOL
SUPER^.EventsDefinition ();

THIS^.SetText (eLocation := E_BaseLocation.pl, wsDescription	:= "Błąd uruchomienia zasilania - brak zgody od safety - BRAK SS1");
THIS^.SetText (eLocation := E_BaseLocation.en, wsDescription	:= "");
THIS^.SetText (eLocation := E_BaseLocation.de, wsDescription	:= "");
THIS^.AddEvent (
	bIgnoreRepetitions			:= TRUE,
	eEventCategory				:= E_BaseEvents_Category.Error,
	bConfirm					:= FALSE,
	stDescription				:= THIS^.GetTexts ()
);
THIS^.SetText (eLocation := E_BaseLocation.pl, wsDescription	:= "Błąd uruchomienia zasilania - brak zgody od safety - BRAK STO");
THIS^.SetText (eLocation := E_BaseLocation.en, wsDescription	:= "");
THIS^.SetText (eLocation := E_BaseLocation.de, wsDescription	:= "");
THIS^.AddEvent (
	bIgnoreRepetitions			:= TRUE,
	eEventCategory				:= E_BaseEvents_Category.Error,
	bConfirm					:= FALSE,
	stDescription				:= THIS^.GetTexts ()
);
END_METHOD

(*			
	RafalOS
	Rafał Osajda		27.03.2025		TC 4024.66
	Obsluga bledow sprawdzanie czy jakis blad sie nei pojawil i ustawienie stanu lub wylaczenie
*)
METHOD PUBLIC ExecuteEveryCycle_Error
VAR
	iI				: INT;
END_VAR
SUPER^.ExecuteEveryCycle_Error ();

FOR iI := 1 TO TO_INT (THIS^.uiNumberOfComponents) DO
	THIS^.arrComponent [iI].ExecuteEveryCycle_Error ();
END_FOR
END_METHOD

(*			
	RafalOS
	Rafał Osajda		27.03.2025		TC 4024.66
	Wywolanie co cykl operacji 
*)
METHOD PUBLIC ExecuteEveryCycle_Operation
VAR
	iI			: INT;
	bError		: BOOL;
END_VAR
SUPER^.ExecuteEveryCycle_Operation ();

FOR iI := 1 TO TO_INT (THIS^.uiNumberOfComponents) DO
	THIS^.arrComponent [iI].ExecuteEveryCycle_Operation ();
END_FOR


(* 	Zasilanie	*)
IF (THIS^.stPower.cmdTurnOn.OperationExecute ()) THEN
	bError				:= FALSE;
	IF (NOT THIS^.itfSS1.GetFlag ()) THEN
		//blad 
		THIS^.EventSetActive (iNumber := 1);
		bError			:= TRUE;
	END_IF
	IF (NOT THIS^.itfSTO.GetFlag ()) THEN
		//blad
		THIS^.EventSetActive (iNumber := 2);
		bError			:= TRUE;
	END_IF
	IF (NOT bError) THEN
		THIS^.stPower.cmdTurnOn.Operation (bIN		:= THIS^.PowerOnCycle ());
		IF (THIS^.EventIsActive (iNumber := 1)) THEN
			THIS^.EventSetInactive (iNumber := 1);
		END_IF
		IF (THIS^.EventIsActive (iNumber := 2)) THEN
			THIS^.EventSetInactive (iNumber := 2);
		END_IF
	ELSE
		THIS^.stPower.cmdTurnOn.Abort ();
	END_IF
END_IF
IF (THIS^.stPower.cmdTurnOff.OperationExecute ()) THEN
	THIS^.stPower.cmdTurnOff.Operation (bIN	:= THIS^.PowerOffCycle ());
END_IF
(*	Bazowanie	*)
IF (THIS^.stHoming.cmdExecute.OperationExecute ()) THEN
	THIS^.stHoming.cmdExecute.Operation (bIN	:= THIS^.HomingCycleInternal ());
END_IF
END_METHOD

(*			
	RafalOS
	Rafał Osajda		27.03.2025		TC 4024.66
	Aktualizacja flag 
*)
METHOD PUBLIC ExecuteEveryCycle_Status
VAR
	iI				: INT;
END_VAR
SUPER^.ExecuteEveryCycle_Status ();

FOR iI := 1 TO TO_INT (THIS^.uiNumberOfComponents) DO
	THIS^.arrComponent [iI].ExecuteEveryCycle_Status ();
END_FOR
END_METHOD

(*			
	RafalOS
	Rafał Osajda		27.03.2025		TC 4024.66
	Testowanie czy nei pojawil sie jakis rozkaz i uruchomienie odpowiednich operacji
*)
METHOD PUBLIC ExecuteEveryCycle_Test
VAR
	iI				: INT;
END_VAR
SUPER^.ExecuteEveryCycle_Test ();

FOR iI := 1 TO TO_INT (THIS^.uiNumberOfComponents) DO
	THIS^.arrComponent [iI].ExecuteEveryCycle_Test ();
END_FOR

THIS^.stPower.cmdTurnOn.Test ();
THIS^.stPower.cmdTurnOff.Test ();

IF (THIS^.stPower.bStatus) THEN
	THIS^.ExecuteEveryCycle_TestWithPower ();
ELSE
	THIS^.ExecuteEveryCycle_TestWithoutPower ();
END_IF
END_METHOD

METHOD PROTECTED ExecuteEveryCycle_TestWithoutPower
VAR_INPUT
END_VAR
THIS^.stHoming.cmdExecute.Abort ();
END_METHOD

METHOD PROTECTED ExecuteEveryCycle_TestWithPower
VAR_INPUT
END_VAR
THIS^.stHoming.cmdExecute.Test ();
END_METHOD

METHOD FB_init : BOOL
VAR_INPUT
	bInitRetains : BOOL; // if TRUE, the retain variables are initialized (warm start / cold start)
	bInCopyCode : BOOL;  // if TRUE, the instance afterwards gets moved into the copy code (online change)
END_VAR
THIS^.stIdentifier.eType			:= E_BaseElementType.eControl;
END_METHOD

METHOD PUBLIC FirstCycle : BOOL
VAR_INPUT
END_VAR
VAR
	bResult			: bool;
	iI				: INT;
END_VAR
bResult				:= SUPER^.FirstCycle ();

FOR iI := 1 TO TO_INT (THIS^.uiNumberOfComponents) DO
	bResult			:= bResult AND THIS^.arrComponent [iI].FirstCycle ();
END_FOR

FirstCycle			:= bResult;
END_METHOD

METHOD GetITFControlElement : ITF_BaseControlElement
VAR_INPUT
END_VAR
GetITFControlElement	:= THIS^;
END_METHOD

METHOD GetITFGroupElement : ITF_BaseGroupElement
VAR_INPUT
END_VAR
GetITFGroupElement	:= null;
END_METHOD

METHOD GetITFTopElement : ITF_BaseTopElement
VAR_INPUT
END_VAR
GetITFTopElement		:= null;
END_METHOD

(*			
	RafalOS
	Rafał Osajda		27.05.2025		TC 4024.66
	Metoda bazowania kontrektnego elementu 
*)
METHOD PROTECTED HomingCycle : BOOL
VAR_INPUT
END_VAR
HomingCycle					:= FALSE;
END_METHOD

(*			
	RafalOS
	Rafał Osajda		27.05.2025		TC 4024.66
	Metoda główna bazowania wywołuje metode przeciążaną Bazowanie_Cykl dziecka
*)
METHOD PRIVATE HomingCycleInternal : BOOL
VAR_INPUT
END_VAR
CASE THIS^.stHoming.cmdExecute.GetStep () OF
0	:
	IF (THIS^.stHoming.bWithoutHoming) THEN	//bazowanie wyłączone true
		THIS^.stHoming.bIsNeeded		:= TRUE;	//ustaw że juz jest wybazowane
		THIS^.stHoming.cmdExecute.SetStepAsFinal ();
	ELSE
		THIS^.stHoming.iElementHomingStep	:= 0;
		THIS^.stHoming.cmdExecute.SetStepINC10 ();
	END_IF
	THIS^.stHoming.bIsNeeded			:= TRUE;
	HomingCycleInternal				:= TRUE;
10	:
	IF (NOT THIS^.HomingCycle ()) THEN
		THIS^.stHoming.cmdExecute.SetStepAsFinal ();
	END_IF
	HomingCycleInternal				:= TRUE;
GVL_BaseConstans.FINISH_STEP	:
	THIS^.stHoming.bIsNeeded			:= FALSE;	//ustaw że juz jest wybazowane
	HomingCycleInternal				:= FALSE;
END_CASE
END_METHOD

(*			
	RafalOS
	Rafał Osajda		27.05.2025		TC 4024.66
	Bazowanie w toku
*)
METHOD PUBLIC HomingGetBusy : BOOL
VAR_INPUT
END_VAR
HomingGetBusy		:= THIS^.stHoming.cmdExecute.IsBusy ();
END_METHOD

(*			
	RafalOS
	Rafał Osajda		31.03.2025		TC 4024.66
	Flaga że w tej sesji pracy maszyny element został już wybazowany
*)
METHOD PUBLIC HomingGetDone : BOOL
VAR_INPUT
END_VAR
HomingGetDone	:= THIS^.stHoming.cmdExecute.IsDone ();
END_METHOD

(*			
	RafalOS
	Rafał Osajda		11.04.2025		TC 4024.66
	Zwraca czy bazowanie jest potrzebne
*)
METHOD PUBLIC HomingGetIsNeeded : BOOL
VAR_INPUT
END_VAR
HomingGetIsNeeded			:= THIS^.stHoming.bIsNeeded;
END_METHOD

(*			
	RafalOS
	Rafał Osajda		11.04.2025		TC 4024.66
	Ustawia czy element jest ma być bazowany czy nie
*)
METHOD PUBLIC HomingSetWithoutHoming : BOOL
VAR_INPUT
	bIN			: BOOL;
END_VAR
THIS^.stHoming.bWithoutHoming			:= bIN;
END_METHOD

(*			
	RafalOS
	Rafał Osajda		27.05.2025		TC 4024.66
	Uruchomienie metody bazowania
*)
METHOD PUBLIC HomingStart
VAR_INPUT
END_VAR
THIS^.stHoming.cmdExecute.Execute ();
END_METHOD

(*			
	RafalOS
	Rafał Osajda		30.04.2025		TC 4024.66
	Zwraca czy element jest czymś zajety
*)
METHOD PUBLIC IsDoNothing : BOOL
IsDoNothing				:= THIS^.bDoNothing;
END_METHOD

(*			
	RafalOS
	Rafał Osajda		30.04.2025		TC 4024.66
	Zwraca czy element jest w pozycji 0 - referencyjnej
*)
METHOD PUBLIC IsPosition0 : BOOL
IsPosition0				:= THIS^.bPosition0;
END_METHOD

METHOD PUBLIC IsValidCommonData : BOOL
VAR_INPUT
END_VAR

VAR
	bResult: BOOL;
	iI: INT;
END_VAR
bResult						:= SUPER^.IsValidCommonData ();

FOR iI := 1 TO TO_INT (THIS^.uiNumberOfComponents) DO
	bResult					:= bResult AND THIS^.arrComponent [iI].IsValidCommonData ();
END_FOR

IsValidCommonData			:= bResult;
END_METHOD

(*			
	RafalOS
	Rafał Osajda		07.10.2025		TC 4024.66
	Dodpisywanie się do listy logera
*)
METHOD PUBLIC JoinTheLogger : BOOL
VAR_INPUT
END_VAR

VAR
	bResult: BOOL;
	iI: INT;
END_VAR
bResult			:= SUPER^.JoinTheLogger ();

FOR iI := 1 TO  TO_INT (THIS^.uiNumberOfComponents) DO
	bResult 	:= bResult AND THIS^.arrComponent [iI].JoinTheLogger ();
END_FOR

JoinTheLogger	:= bResult;
END_METHOD

METHOD PUBLIC LinkCommonData : BOOL
VAR_INPUT
	stCommonData				: REFERENCE TO ST_BaseCommonData;
END_VAR
VAR
	bResult						: BOOL;
	iI: INT;
END_VAR
bResult							:= SUPER^.LinkCommonData (stCommonData := stCommonData);

FOR iI := 1 TO TO_INT (THIS^.uiNumberOfComponents) DO
	bResult := bResult AND THIS^.arrComponent [iI].LinkCommonData (stCommonData := stCommonData);
END_FOR

LinkCommonData					:= bResult;
END_METHOD

METHOD PUBLIC LinkSS1 : BOOL
VAR_INPUT
	fbSS1			: ITF_BaseFlagGet;
END_VAR
THIS^.itfSS1		:= fbSS1;

LinkSS1				:= THIS^.itfSS1 <> 0;
END_METHOD

METHOD PUBLIC LinkSTO : BOOL
VAR_INPUT
	fbSTO			: ITF_BaseFlagGet;
END_VAR
THIS^.itfSTO		:= fbSTO;

LinkSTO				:= THIS^.itfSTO <> 0;
END_METHOD

(*			
	RafalOS
	Rafał Osajda		31.03.2025		TC 4024.66
	Zwraca status zasilania	
*)
METHOD PUBLIC PowerGetStatus : BOOL
VAR_INPUT
END_VAR
PowerGetStatus			:= THIS^.stPower.bStatus;
END_METHOD

(*			
	RafalOS
	Rafał Osajda		13.10.2025		TC 4024.66
	Podstawowy cykl wyłączania zasilania. Dla Specyficznych urządzeń przeciążyć
*)
METHOD PROTECTED PowerOffCycle : BOOL
THIS^.stPower.bStatus		:= FALSE;
PowerOffCycle				:= FALSE;
END_METHOD

(*			
	RafalOS
	Rafał Osajda		13.10.2025		TC 4024.66
	Podstawowy cykl włączania zasilania. Dla Specyficznych urządzeń przeciążyć
*)
METHOD PROTECTED PowerOnCycle : BOOL
THIS^.stPower.bStatus		:= TRUE;
PowerOnCycle				:= FALSE;
END_METHOD

(*			
	RafalOS
	Rafał Osajda		31.03.2025		TC 4024.66
	Wyłączenie zasilania
*)
METHOD PUBLIC PowerTurnOff : BOOL
VAR_INPUT
END_VAR
THIS^.stPower.cmdTurnOff.Execute ();
END_METHOD

METHOD PUBLIC PowerTurnOffDone : BOOL
VAR_INPUT
END_VAR
PowerTurnOffDone		:= THIS^.stPower.cmdTurnOff.IsDone ();
END_METHOD

METHOD PUBLIC PowerTurnOffInProgress : BOOL
VAR_INPUT
END_VAR
PowerTurnOffInProgress			:= THIS^.stPower.cmdTurnOff.IsBusy ();
END_METHOD

(*			
	RafalOS
	Rafał Osajda		31.03.2025		TC 4024.66
	Uruchomienie zasialania
*)
METHOD PUBLIC PowerTurnOn
VAR_INPUT
END_VAR
THIS^.stPower.cmdTurnOn.Execute ();
END_METHOD

METHOD PUBLIC PowerTurnOnDone : BOOL
VAR_INPUT
END_VAR
PowerTurnOnDone		:= THIS^.stPower.cmdTurnOn.IsDone ();
END_METHOD

METHOD PUBLIC PowerTurnOnInProgress : BOOL
VAR_INPUT
END_VAR
PowerTurnOnInProgress		:= THIS^.stPower.cmdTurnOn.IsBusy ();
END_METHOD

METHOD PROTECTED ResetOperation : BOOL
VAR
	bResult				: BOOL;
END_VAR
bResult					:= SUPER^.ResetOperation ();

THIS^.stHoming.bIsNeeded	:= TRUE;
THIS^.stHoming.cmdExecute.Abort ();
THIS^.stHoming.iChildHomingStep	:= 0;
THIS^.stHoming.iElementHomingStep	:= 0;

ResetOperation			:= FALSE OR bResult;
END_METHOD

METHOD PUBLIC SetCode
VAR_INPUT
	sCode							: STRING;
	sAdd							: STRING;
END_VAR
VAR
	sItemCode						: STRING;
	iI								: INT;
	sComponentCode					: STRING;
END_VAR
sItemCode		:=  CreateElementCode (sParentCode := sCode, sAdd := sAdd);
SUPER^.SetCode (sCode := sItemCode, sAdd := '');

FOR iI := 1 TO TO_INT (THIS^.uiNumberOfComponents) DO
	sComponentCode	:= CreateElementCode (sParentCode := sItemCode, sAdd := TO_STRING (iI));
	THIS^.arrComponent [iI].SetCode (sCode	:= sComponentCode, sAdd := '');
END_FOR
END_METHOD

(*			
	RafalOS
	Rafał Osajda		03.10.2025		TC 4024.66
	nadawanie unikalnych ID dla zdarzeń
*)
METHOD PUBLIC SetEventsIDs : UINT
VAR_INPUT
	uiNewID		: UINT;
END_VAR
VAR
	iI			: INT;
	uiLastID	: UINT;
END_VAR
uiLastID		:= SUPER^.SetEventsIDs (uiNewID	:= uiNewID);

FOR iI := 1 TO TO_INT (THIS^.uiNumberOfComponents) DO 
	uiLastID			:= THIS^.arrComponent [iI].SetEventsIDs (uiNewID	:= uiLastID);
END_FOR
SetEventsIDs				:= uiLastID;
END_METHOD

METHOD PUBLIC SetID : UINT
VAR_INPUT
	uiID					: UINT;
END_VAR
VAR
	uiLastID				: UINT;
	iI						: INT;
END_VAR
uiLastID				:= SUPER^.SetID (uiID	:= uiID);

FOR iI := 1 TO TO_INT (THIS^.uiNumberOfComponents) DO 
	uiLastID			:= THIS^.arrComponent [iI].SetID (uiID	:= uiLastID + 1);
END_FOR
SetID					:= uiLastID;
END_METHOD

END_FUNCTION_BLOCK

// ---- FUNs/CreateElementCode.TcPOU
(*			RafalOS
	Rafał Osajda		16.10.2024		TC 4026.11		wer. 0.0.0.1
	Utworzenie kodu elementu 
*)
FUNCTION CreateElementCode : STRING
VAR_INPUT
	sParentCode					: STRING;
	sAdd						: STRING;
END_VAR
VAR
	arrSegments					: ARRAY [0..GVL_BaseConstans.MAX_NESTING_LEVEL] OF STRING;
	iI							: INT;
	iDotPosition				: INT;
	sCodeResult					: STRING;
END_VAR

IF (LEN (STR := sParentCode) > 0) THEN
	arrSegments [0]				:= sParentCode;
	FOR iI := 1 TO TO_INT (GVL_BaseConstans.MAX_NESTING_LEVEL) DO
		iDotPosition			:= find (STR1 := arrSegments [0], STR2 := '.');
		IF (iDotPosition = 0) THEN
			arrSegments [iI]	:= arrSegments [0];
			EXIT;
		ELSE
			arrSegments [iI]	:= LEFT (STR := arrSegments [0], SIZE := iDotPosition - 1);
			arrSegments [0]		:= delete (STR := arrSegments [0], POS := 1, LEN := iDotPosition);
		END_IF
	END_FOR
END_IF
FOR iI := 1 TO TO_INT (GVL_BaseConstans.MAX_NESTING_LEVEL) DO
	IF (arrSegments [iI] = '0' OR arrSegments [iI] = '') THEN
		arrSegments [iI] := sAdd;
		sAdd			:= '0';
	END_IF
	sCodeResult			:= CONCAT (STR1 := sCodeResult, STR2 := arrSegments [iI]);
	IF (iI < TO_INT (GVL_BaseConstans.MAX_NESTING_LEVEL)) THEN
		sCodeResult		:= CONCAT (STR1 := sCodeResult, STR2 := '.');
	END_IF
END_FOR

CreateElementCode							:= sCodeResult;

END_FUNCTION

// ---- POUs/A06_FB_BaseGroupElement/FB_BaseGroupElement.TcPOU
(*			
	RAFALOS
	Rafał Osajda		19.09.2025		TC 4024.66
	FB Bazowy dla wszystkich elementów złożonych
*)
FUNCTION_BLOCK FB_BaseGroupElement EXTENDS FB_BaseControlElement IMPLEMENTS ITF_BaseGroupElement, ITF_BaseGroupElement_HMI_Connector,
 		ITF_BaseMessengerRecipient, ITF_BaseMessengerSender
VAR
	arrControlElement			: ARRAY [1..GVL_BaseConstans.MAX_ITEM_PER_ELEMENT] OF ITF_BaseControlElement;
	uiNumberOfControlElement	: UINT;
	itfCommunicator				: ITF_BaseCommunicator;
END_VAR

METHOD PROTECTED AddControlElement : BOOL
VAR_INPUT
	itfControlElement		: ITF_BaseControlElement;
END_VAR
IF (THIS^.uiNumberOfControlElement + 1 <= GVL_BaseConstans.MAX_ITEM_PER_ELEMENT) THEN
	THIS^.uiNumberOfControlElement		:= THIS^.uiNumberOfControlElement + 1;
	THIS^.arrControlElement [THIS^.uiNumberOfControlElement]	:= itfControlElement;
	AddControlElement			:= TRUE;
ELSE
	;//zwrocenie zbyt dużo komponentow
END_IF
END_METHOD

METHOD PUBLIC ConfirmReceipt : BOOL
VAR_INPUT
	sText: STRING;
END_VAR
ConfirmReceipt	:= THIS^.itfCommunicator.ReceiveDataConfirm (sText := sText, itfRecipient := THIS^);
END_METHOD

(*			
	RafalOS
	Rafał Osajda		27.03.2025		TC 4024.66
	Obsluga bledow sprawdzanie czy jakis blad sie nei pojawil i ustawienie stanu lub wylaczenie
*)
METHOD PUBLIC ExecuteEveryCycle_Error
VAR
	iI					: INT;
END_VAR
SUPER^.ExecuteEveryCycle_Error ();

FOR iI := 1 TO TO_INT (THIS^.uiNumberOfControlElement) DO
	THIS^.arrControlElement [iI].ExecuteEveryCycle_Error ();
END_FOR
END_METHOD

(*			
	RafalOS
	Rafał Osajda		27.03.2025		TC 4024.66
	Wywolanie co cykl operacji 
*)
METHOD PUBLIC ExecuteEveryCycle_Operation
VAR
	iI				: INT;
END_VAR
SUPER^.ExecuteEveryCycle_Operation ();

FOR iI := 1 TO TO_INT (THIS^.uiNumberOfControlElement) DO
	THIS^.arrControlElement [iI].ExecuteEveryCycle_Operation ();
END_FOR
END_METHOD

(*			
	RafalOS
	Rafał Osajda		27.03.2025		TC 4024.66
	Aktualizacja flag 
*)
METHOD PUBLIC ExecuteEveryCycle_Status
VAR
	iI				: INT;
END_VAR
SUPER^.ExecuteEveryCycle_Status ();

FOR iI := 1 TO TO_INT (THIS^.uiNumberOfControlElement) DO
	THIS^.arrControlElement [iI].ExecuteEveryCycle_Status ();
END_FOR
END_METHOD

(*			
	RafalOS
	Rafał Osajda		27.03.2025		TC 4024.66
	Testowanie czy nei pojawil sie jakis rozkaz i uruchomienie odpowiednich operacji
*)
METHOD PUBLIC ExecuteEveryCycle_Test
VAR
	iI			: INT;
END_VAR
SUPER^.ExecuteEveryCycle_Test ();

FOR iI := 1 TO TO_INT (THIS^.uiNumberOfControlElement) DO
	THIS^.arrControlElement [iI].ExecuteEveryCycle_Test ();
END_FOR
END_METHOD

METHOD FB_init : BOOL
VAR_INPUT
	bInitRetains : BOOL; // if TRUE, the retain variables are initialized (warm start / cold start)
	bInCopyCode : BOOL;  // if TRUE, the instance afterwards gets moved into the copy code (online change)
END_VAR
THIS^.stIdentifier.eType			:= E_BaseElementType.eGroup;
END_METHOD

METHOD PUBLIC FirstCycle : BOOL
VAR_INPUT
END_VAR
VAR
	bResult			: bool;
	iI				: INT;
END_VAR
bResult				:= SUPER^.FirstCycle ();

FOR iI := 1 TO TO_INT (THIS^.uiNumberOfControlElement) DO
	bResult			:= bResult AND THIS^.arrControlElement [iI].FirstCycle ();
END_FOR

FirstCycle			:= bResult;
END_METHOD

METHOD GetITFGroupElement : ITF_BaseGroupElement
VAR_INPUT
END_VAR
GetITFGroupElement	:= THIS^;
END_METHOD

METHOD GetITFTopElement : ITF_BaseTopElement
VAR_INPUT
END_VAR
GetITFTopElement		:= null;
END_METHOD

(*			
	RafalOS
	Rafał Osajda		27.05.2025		TC 4024.66
	Metoda bazowania kontrektnego elementu 
*)
METHOD PROTECTED HomingCycle : BOOL
VAR
	iI			: INT;
END_VAR
CASE THIS^.stHoming.iElementHomingStep OF
0	:
	FOR iI := 1 TO TO_INT (THIS^.uiNumberOfControlElement) DO
		THIS^.arrControlElement [iI].HomingStart ();
	END_FOR
	THIS^.stHoming.iElementHomingStep	:= THIS^.stHoming.iElementHomingStep + 10;
	HomingCycle							:= TRUE;
10	:
	THIS^.stHoming.iElementHomingStep	:= THIS^.stHoming.iElementHomingStep + 10;
	HomingCycle							:= TRUE;
20	:
	IF (THIS^.HomingGetDone ()) THEN
		THIS^.stHoming.iElementHomingStep 	:= GVL_BaseConstans.FINISH_STEP;
	END_IF	
	HomingCycle							:= TRUE;
GVL_BaseConstans.FINISH_STEP :
	HomingCycle							:= FALSE;
END_CASE
END_METHOD

(*			
	RafalOS
	Rafał Osajda		31.03.2025		TC 4024.66
	Flaga że w tej sesji pracy maszyny element został już wybazowany
*)
METHOD PUBLIC HomingGetDone : BOOL
VAR
	iI				: INT;
	btmpHomingDone	: BOOL;
END_VAR
btmpHomingDone		:= TRUE;
FOR iI := 1 TO TO_INT (THIS^.uiNumberOfControlElement) DO
	btmpHomingDone	:= btmpHomingDone AND THIS^.arrControlElement [iI].HomingGetDone ();
	IF (NOT btmpHomingDone) THEN
		EXIT;
	END_IF
END_FOR
HomingGetDone		:= btmpHomingDone;
END_METHOD

(*			
	RafalOS
	Rafał Osajda		11.04.2025		TC 4024.66
	Zwraca czy bazowanie jest potrzebne
*)
METHOD PUBLIC HomingGetIsNeeded : BOOL
VAR
	btmpHomingIsNeeded	: BOOL := FALSE;
	iI					: INT;
END_VAR
FOR iI := 1 TO TO_INT (THIS^.uiNumberOfControlElement) DO
	btmpHomingIsNeeded	:= btmpHomingIsNeeded OR THIS^.arrControlElement [iI].HomingGetIsNeeded ();
	IF (btmpHomingIsNeeded) THEN
		EXIT;
	END_IF
END_FOR
HomingGetIsNeeded		:= btmpHomingIsNeeded;
END_METHOD

(*			
	RafalOS
	Rafał Osajda		30.04.2025		TC 4024.66
	Zwraca czy element jest czymś zajety
*)
METHOD PUBLIC IsDoNothing : BOOL
VAR
	iI				: INT;
	btmpDoNothing	: BOOL := TRUE;
END_VAR
FOR iI := 1 TO TO_INT (THIS^.uiNumberOfControlElement) DO
	btmpDoNothing		:= btmpDoNothing AND THIS^.arrControlElement [iI].IsDoNothing ();
	IF (NOT btmpDoNothing) THEN
		EXIT;
	END_IF
END_FOR
THIS^.bDoNothing		:= btmpDoNothing;
IsDoNothing			:= btmpDoNothing;
END_METHOD

(*			
	RafalOS
	Rafał Osajda		30.04.2025		TC 4024.66
	Zwraca czy element jest w pozycji 0 - referencyjnej
*)
METHOD PUBLIC IsPosition0 : BOOL
VAR
	iI					: INT;
	btmpPosition0		: BOOL;
END_VAR
FOR iI := 1 TO TO_INT (THIS^.uiNumberOfControlElement) DO
	btmpPosition0		:= btmpPosition0 AND THIS^.arrControlElement [iI].IsPosition0 ();
	IF (NOT btmpPosition0) THEN
		EXIT;
	END_IF
END_FOR
THIS^.bPosition0		:= btmpPosition0;
IsPosition0			:= btmpPosition0;
END_METHOD

METHOD PUBLIC IsValidCommonData : BOOL
VAR_INPUT
END_VAR

VAR
	bResult: BOOL;
	iI: INT;
END_VAR
bResult						:= SUPER^.IsValidCommonData ();

FOR iI := 1 TO TO_INT (THIS^.uiNumberOfControlElement) DO
	bResult					:= bResult AND THIS^.arrControlElement [iI].IsValidCommonData ();
END_FOR

IsValidCommonData			:= bResult;
END_METHOD

(*			
	RafalOS
	Rafał Osajda		07.10.2025		TC 4024.66
	Dodpisywanie się do listy logera
*)
METHOD PUBLIC JoinTheLogger : BOOL
VAR_INPUT
END_VAR

VAR
	bResult: BOOL;
	iI: INT;
END_VAR
bResult			:= SUPER^.JoinTheLogger ();

FOR iI := 1 TO  TO_INT (THIS^.uiNumberOfControlElement) DO
	bResult 	:= bResult AND THIS^.arrControlElement [iI].JoinTheLogger ();
END_FOR

JoinTheLogger	:= bResult;
END_METHOD

METHOD PUBLIC LinkCommonData : BOOL
VAR_INPUT
	stCommonData				: REFERENCE TO ST_BaseCommonData;
END_VAR
VAR
	bResult						: BOOL;
	iI: INT;
END_VAR
bResult							:= SUPER^.LinkCommonData (stCommonData := stCommonData);

FOR iI := 1 TO TO_INT (THIS^.uiNumberOfControlElement) DO
	bResult := bResult AND THIS^.arrControlElement [iI].LinkCommonData (stCommonData := stCommonData);
END_FOR

LinkCommonData					:= bResult;
END_METHOD

METHOD PUBLIC LinkCommunicator : BOOL
VAR_INPUT
	fbCommunicator				: ITF_BaseCommunicator;
END_VAR
THIS^.itfCommunicator			:= fbCommunicator;
IF (THIS^.itfCommunicator <> 0) THEN
	LinkCommunicator			:= TRUE;
END_IF
END_METHOD

METHOD PUBLIC LinkSS1 : BOOL
VAR_INPUT
	fbSS1			: ITF_BaseFlagGet;
END_VAR

VAR
	bresult: BOOL;
	iI: INT;
END_VAR
bresult				:= SUPER^.LinkSS1 (fbSS1 := fbSS1);

FOR iI := 1 TO TO_INT (THIS^.uiNumberOfControlElement) DO
	bresult			:= bresult AND THIS^.arrControlElement [iI].LinkSS1 (fbSS1	:= fbSS1);
END_FOR

LinkSS1				:= bresult;
END_METHOD

METHOD PUBLIC LinkSTO : BOOL
VAR_INPUT
	fbSTO			: ITF_BaseFlagGet;
END_VAR

VAR
	bresult: BOOL;
	iI: INT;
END_VAR
bresult				:= SUPER^.LinkSTO (fbSTO := fbSTO);

FOR iI := 1 TO TO_INT (THIS^.uiNumberOfControlElement) DO
	bresult			:= bresult AND THIS^.arrControlElement [iI].LinkSTO (fbSTO	:= fbSTO);
END_FOR

LinkSTO				:= bresult;
END_METHOD

METHOD PROTECTED PowerOffCycle : BOOL
VAR
	iI							: INT;
	bPowerStatus			: BOOL;
END_VAR
CASE stPower.cmdTurnOff.GetStep () OF
0	:
	FOR iI := 1 TO TO_INT (THIS^.uiNumberOfControlElement) DO
		THIS^.arrControlElement [iI].PowerTurnOff ();
	END_FOR
	THIS^.stPower.cmdTurnOff.SetStepINC10 ();
	PowerOffCycle			:= TRUE;
10	:
	bPowerStatus			:= FALSE;
	FOR iI := 1 TO TO_INT (THIS^.uiNumberOfControlElement) DO
		bPowerStatus		:= bPowerStatus OR THIS^.arrControlElement [iI].PowerGetStatus ();
		IF (bPowerStatus) THEN
			EXIT;
		END_IF
	END_FOR	
	IF (NOT bPowerStatus) THEN
		THIS^.stPower.bStatus	:= FALSE;
		THIS^.stPower.cmdTurnOff.SetStepAsFinal ();
	ELSE
		PowerOffCycle			:= TRUE;
	END_IF	
END_CASE
END_METHOD

METHOD PROTECTED PowerOnCycle : BOOL
VAR
	iI						: INT;
	bPowerStatus		: BOOL;
END_VAR
CASE stPower.cmdTurnOn.GetStep () OF
0	:
	FOR iI := 1 TO TO_INT (THIS^.uiNumberOfControlElement) DO
		THIS^.arrControlElement [iI].PowerTurnOn ();
	END_FOR
	THIS^.stPower.cmdTurnOn.SetStepINC10 ();
	PowerOnCycle				:= TRUE;
10	:
	bPowerStatus			:= TRUE;
	FOR iI := 1 TO TO_INT (THIS^.uiNumberOfControlElement) DO
		bPowerStatus		:= bPowerStatus AND THIS^.arrControlElement [iI].PowerGetStatus ();
		IF (NOT bPowerStatus) THEN
			EXIT;
		END_IF
	END_FOR	
	IF (bPowerStatus) THEN
		THIS^.stPower.bStatus	:= TRUE;
		THIS^.stPower.cmdTurnOn.SetStepAsFinal ();
		PowerOnCycle			:= FALSE;
	ELSE
		PowerOnCycle			:= TRUE;
	END_IF	
END_CASE
END_METHOD

METHOD PUBLIC Receive_BOOL : BOOL
VAR_INPUT
	sText		: STRING;
END_VAR
VAR_OUTPUT
	bValue		: BOOL;	
END_VAR
Receive_BOOL			:= THIS^.itfCommunicator.ReceiveData_BOOL (sText := sText, itfRecipient := THIS^, bValue => bValue);
END_METHOD

METHOD PUBLIC Receive_REAL : BOOL
VAR_INPUT
	sText		: STRING;
END_VAR
VAR_OUTPUT
	rValue		: REAL;	
END_VAR
Receive_REAL			:=  THIS^.itfCommunicator.ReceiveData_REAL (sText := sText, itfRecipient := THIS^, rValue => rValue);
END_METHOD

METHOD PROTECTED ResetOperation : BOOL
VAR
	bResult				: BOOL;
END_VAR
bResult					:= SUPER^.ResetOperation ();


ResetOperation			:= FALSE OR bResult;
END_METHOD

METHOD Send_BOOL : BOOL
VAR_INPUT
	sText				: STRING;
END_VAR
Send_BOOL		:= THIS^.itfCommunicator.SendData_BOOL (sText := sText, itfSender := THIS^);
END_METHOD

METHOD Send_REAL : BOOL
VAR_INPUT
	sText		: STRING;
	rValue		: REAL;
END_VAR
Send_REAL			:= THIS^.itfCommunicator.SendData_REAL (sText := sText, rValue := rValue, itfSender := THIS^);
END_METHOD

METHOD PUBLIC SetCode
VAR_INPUT
	sCode							: STRING;
	sAdd							: STRING;
END_VAR
VAR
	sItemCode						: STRING;
	iI								: INT;
	sParentCode						: STRING;
	arrSegment						: ARRAY [0..GVL_BaseConstans.MAX_NESTING_LEVEL] OF STRING;
	iDotPosition					: INT;
	iLast							: INT;
	
END_VAR
//sKodRodzica	:=  UtworzKodElementu (sKodRodzica := sKod, sDopisz := TO_STRING (THIS^.zwrocID ()));
SUPER^.SetCode (sCode := sCode, sAdd := sAdd);
sParentCode						:= THIS^.GetCode ();

IF (THIS^.uiNumberOfComponents > 0) THEN
	arrSegment [0]				:= THIS^.arrComponent [THIS^.uiNumberOfComponents].GetCode ();
	FOR iI := 1 TO TO_INT (GVL_BaseConstans.MAX_NESTING_LEVEL) DO
		iDotPosition			:= find (STR1 := arrSegment [0], STR2 := '.');
		IF (iDotPosition = 0) THEN
			arrSegment [iI]	:= arrSegment [0];
			EXIT;
		ELSE
			arrSegment [iI]		:= Tc2_Standard.LEFT (STR := arrSegment [0], SIZE := iDotPosition - 1);
			arrSegment [0]		:= Tc2_Standard.DELETE (STR := arrSegment [0], POS := 1, LEN := iDotPosition);
		END_IF
	END_FOR
	FOR iI := 0 TO TO_INT (GVL_BaseConstans.MAX_NESTING_LEVEL) - 1 DO
		IF (TO_INT (arrSegment [TO_INT (GVL_BaseConstans.MAX_NESTING_LEVEL) - iI]) <> 0 ) THEN
			iLast			:= TO_INT (arrSegment [TO_INT (GVL_BaseConstans.MAX_NESTING_LEVEL) - iI]);
			EXIT;
		END_IF
	END_FOR
END_IF

FOR iI := 1 TO TO_INT (THIS^.uiNumberOfControlElement) DO
//	sKodKomponentu	:= UtworzKodElementu (sKodRodzica := sKod, sDopisz := TO_STRING (iI));
	THIS^.arrControlElement [iI].SetCode (sCode	:= sParentCode, sAdd := TO_STRING (iI + iLast));
END_FOR
END_METHOD

(*			
	RafalOS
	Rafał Osajda		03.10.2025		TC 4024.66
	nadawanie unikalnych ID dla zdarzeń
*)
METHOD PUBLIC SetEventsIDs : UINT
VAR_INPUT
	uiNewID		: UINT;
END_VAR
VAR
	iI			: INT;
	uiLastID	: UINT;
END_VAR
uiLastID		:= SUPER^.SetEventsIDs (uiNewID	:= uiNewID);

FOR iI := 1 TO TO_INT (THIS^.uiNumberOfControlElement) DO 
	uiLastID			:= THIS^.arrControlElement [iI].SetEventsIDs (uiNewID	:= uiLastID);
END_FOR
SetEventsIDs				:= uiLastID;
END_METHOD

METHOD PUBLIC SetID : UINT
VAR_INPUT
	uiID					: UINT;
END_VAR
VAR
	uiLastID				: UINT;
	iI						: INT;
END_VAR
uiLastID				:= SUPER^.SetID (uiID	:= uiID);

FOR iI := 1 TO TO_INT (THIS^.uiNumberOfControlElement) DO 
	uiLastID			:= THIS^.arrControlElement [iI].SetID (uiID	:= uiLastID + 1);
END_FOR
SetID					:= uiLastID;
END_METHOD

END_FUNCTION_BLOCK

// ---- POUs/B02_Recipes/FB_BaseRecipe.TcPOU
(*			
	RafalOS
	Rafał Osajda		28.02.2025		TC 4026.13		wer. 0.0.0.1
	Obsługa receptur
*)
FUNCTION_BLOCK FB_BaseRecipe EXTENDS FB_Base IMPLEMENTS ITF_BaseRecipe, ITF_BaseCreatingTemplateMethod, ITF_BaseRecipe_HMI_Connector
VAR
	iNumberToChoose				: INT;		//numer wybranej
	arritfCreatingRecipe		: ARRAY [1..GVL_BaseConstans.MAX_NUMBER_OF_TEMPLATES] OF ITF_BaseCreateTemplateOfRecipe;
	uiNumberOfCreatingRecipe	: UINT;		//ilosc fb dla tworzenia receptur
END_VAR
VAR PERSISTENT
	arrTemplates				: ARRAY [1..GVL_BaseConstans.MAX_NUMBER_OF_TEMPLATES] OF ST_BaseRecipe;	//szablony
	arrRecipes					: ARRAY [1..GVL_BaseConstans.MAX_NUMBER_OF_RECIPES] OF ST_BaseRecipe;	//receptury
	uiNumberOfTemplates			: UINT;			//ilość dodanych szablonów
	uiNumberOfRecipes			: UINT;			//ilość dodanych receptur
	uiChosen					: UINT;			//numer wybranej receptruy		
	stChosen					: ST_BaseRecipe;	//kopia wybranej recepury kopiowana w momencie wyboru, zmiany w recepturze bazowej nie jest przepisywana automatycznia
END_VAR

(*			
	RafalOS
	Rafał Osajda		25.10.2025		TC 4024.66
	Dodawanie składnika do szablonu
*)
METHOD PUBLIC AddIngredientToTemplate : BOOL
VAR_INPUT
	uiNumber		: UINT;
	stIngredient	: ST_BaseDescriptor;
END_VAR
IF (THIS^.arrTemplates [uiNumber].uiNumber + 1 <= GVL_BaseConstans.MAX_NUMBER_Of_INGREDIENTS) THEN
	THIS^.arrTemplates [uiNumber].uiNumber			:= THIS^.arrTemplates [uiNumber].uiNumber + 1;
	THIS^.arrTemplates [uiNumber].arrIngredient [THIS^.arrTemplates [uiNumber].uiNumber]	:= stIngredient;
//	THIS^.arrSzablony [uiNumer].arrSkladnik [THIS^.arrSzablony [uiNumer].uiIlosc].PowiarzJezyk (fbLokalizacja := THIS^.itfJezyk);
	AddIngredientToTemplate						:= TRUE;
END_IF
END_METHOD

(*			
	RafalOS
	Rafał Osajda		25.10.2025		TC 4024.66
	Dodanie itferfejsu FB dla tworzenia szablonów receptur z programu maszyny
*)
METHOD PUBLIC AddITFToCreateTemplate : BOOL
VAR_INPUT
	fbToCtreateTemplate		: ITF_BaseCreateTemplateOfRecipe;
END_VAR
IF (THIS^.uiNumberOfCreatingRecipe + 1 <= GVL_BaseConstans.MAX_NUMBER_OF_TEMPLATES) THEN
	THIS^.uiNumberOfCreatingRecipe	:= THIS^.uiNumberOfCreatingRecipe + 1;
	THIS^.arritfCreatingRecipe [THIS^.uiNumberOfCreatingRecipe]	:= fbToCtreateTemplate;
	AddITFToCreateTemplate		:= TRUE;
ELSE
	AddITFToCreateTemplate		:= FALSE;
END_IF
END_METHOD

(*			
	RafalOS
	Rafał Osajda		03.03.2025		TC 4026.13		wer. 0.0.0.1
	Kopiuje składniki z wybranej receptury i tworzy nową recepture
*)
METHOD PUBLIC AddRecipeFromRecipe : BOOL
VAR_INPUT
	uiNumberRecipe				: UINT;
	stTexts						: ST_BaseLabel;
END_VAR
IF (THIS^.uiNumberOfRecipes + 1 <= GVL_BaseConstans.MAX_NUMBER_OF_RECIPES) THEN
	THIS^.uiNumberOfRecipes					:= THIS^.uiNumberOfRecipes + 1;
	THIS^.arrRecipes [THIS^.uiNumberOfRecipes]	:= THIS^.arrRecipes [uiNumberRecipe];
	THIS^.arrRecipes [THIS^.uiNumberOfRecipes].stTexts	:= stTexts;
//	THIS^.arrReceptury [THIS^.uiIloscReceptur].fbNazwa.PowiarzJezyk (fbLokalizacja := THIS^.itfJezyk);	
	AddRecipeFromRecipe				:= TRUE;
END_IF
END_METHOD

(*			
	RafalOS
	Rafał Osajda		03.03.2025		TC 4026.13		wer. 0.0.0.1
	Kopiuje składniki z wybranego szablonu i tworzy nową recepture
*)
METHOD PUBLIC AddRecipeFromTemplate : BOOL
VAR_INPUT
	uiNumberTemplates			: UINT;
	stTexts						: ST_BaseLabel;
END_VAR
IF (THIS^.uiNumberOfRecipes + 1 <= GVL_BaseConstans.MAX_NUMBER_OF_RECIPES) THEN
	THIS^.uiNumberOfRecipes					:= THIS^.uiNumberOfRecipes + 1;
	THIS^.arrRecipes [THIS^.uiNumberOfRecipes]	:= THIS^.arrTemplates [uiNumberTemplates];
	THIS^.arrRecipes [THIS^.uiNumberOfRecipes].stTexts	:= stTexts;
//	THIS^.arrReceptury [THIS^.uiIloscReceptur].fbNazwa.PowiarzJezyk (fbLokalizacja := THIS^.itfJezyk);
	AddRecipeFromTemplate				:= TRUE;
END_IF
END_METHOD

(*			
	RafalOS
	Rafał Osajda		25.10.2025		TC 4024.66
	Dodawanie szablonu - metoda wykorzystywana w zewnętrznym FB tworzenia receptur
*)
METHOD PUBLIC AddTemplate : BOOL
VAR_INPUT
	stTexts			: ST_BaseLabel;
END_VAR
IF (THIS^.uiNumberOfTemplates + 1 <= GVL_BaseConstans.MAX_NUMBER_OF_TEMPLATES) THEN
	THIS^.uiNumberOfTemplates := THIS^.uiNumberOfTemplates + 1;
	THIS^.arrTemplates [THIS^.uiNumberOfTemplates].stTexts :=  stTexts;
	THIS^.arrTemplates [THIS^.uiNumberOfTemplates].uiTemplate := THIS^.uiNumberOfTemplates;
	AddTemplate := TRUE;
END_IF
END_METHOD

(*			
	RafalOS
	Rafał Osajda		03.03.2025		TC 4026.13		wer. 0.0.0.1
	Przypisuje do referencji wybraną rtecepture
*)
METHOD PUBLIC Choose : BOOL
VAR_INPUT
	uiNumber				: UINT;
END_VAR
THIS^.stChosen := THIS^.arrRecipes [uiNumber];
THIS^.uiChosen := uiNumber;
END_METHOD

(*			
	RafalOS
	Rafał Osajda		03.06.2025		TC 4024.66
	usuwa referencje do wybranej
*)
METHOD PUBLIC ClearChosen
VAR_INPUT
END_VAR
THIS^.uiChosen := 0;
END_METHOD

(*			
	RafalOS
	Rafał Osajda		25.10.2025		TC 4024.66
	Utworzenie nowych szablonów receptur na podstawie dodanych fb zewnętrznych - wywołanie metody powoduje
	skosowanie dotychczasowych szablonów i receptur
*)
METHOD PUBLIC CreateTemplates : BOOL
VAR_INPUT
END_VAR

VAR
	iI: INT;
END_VAR
THIS^.DeleteRecipes ();
THIS^.DeleteTemplates ();

FOR iI := 1 TO TO_INT (THIS^.uiNumberOfCreatingRecipe) DO
	THIS^.arritfCreatingRecipe [iI].CreateTamplateOfRecipe (itfRecipe := THIS^);
END_FOR
END_METHOD

(*			
	RafalOS
	Rafał Osajda		03.03.2025		TC 4026.13		wer. 0.0.0.1
	
*)
METHOD PUBLIC DeleteRecipe : BOOL
VAR_INPUT
	uiNumber				: uint;
END_VAR
IF (uiNumber > 0 AND uiNumber <= THIS^.uiNumberOfRecipes) THEN

	MEMMOVE (
		destAddr						:= ADR (THIS^.arrRecipes [uiNumber]),
		srcAddr							:= ADR (THIS^.arrRecipes [uiNumber + 1]),
		n								:= SIZEOF (THIS^.arrRecipes [1]) * (GVL_BaseConstans.MAX_NUMBER_OF_RECIPES - (uiNumber))
	);
	THIS^.uiNumberOfRecipes				:= THIS^.uiNumberOfRecipes - 1;
	
	DeleteRecipe			:= TRUE;
END_IF
END_METHOD

(*			
	RafalOS
	Rafał Osajda		30.04.2025		TC 4024.66
	usunięcie wszystkich receptur
*)
METHOD PUBLIC DeleteRecipes : BOOL
VAR_INPUT
END_VAR
MEMSET (
	destAddr			:= ADR (THIS^.arrRecipes),
	fillByte			:= 0,
	n					:= SIZEOF (THIS^.arrRecipes)
);
THIS^.uiNumberOfRecipes 	:= 0;
THIS^.uiChosen			:= 0;
END_METHOD

(*			
	RafalOS
	Rafał Osajda		30.04.2025		TC 4024.66
	usunięcie wszystkich szablonów
*)
METHOD PUBLIC DeleteTemplates : BOOL
VAR_INPUT
END_VAR
MEMSET (
	destAddr			:= ADR (THIS^.arrTemplates),
	fillByte			:= 0,
	n					:= SIZEOF (THIS^.arrTemplates)
);
THIS^.uiNumberOfTemplates 	:= 0;

//THIS^.PowiazJezyk (fbLokalizacja := THIS^.itfJezyk);
END_METHOD

(*			
	RafalOS
	Rafał Osajda		03.03.2025		TC 4026.13		wer. 0.0.0.1
	Zwraca referencje do  receptury
*)
METHOD PUBLIC GetAdressOfRecipe : POINTER TO ST_BaseRecipe
VAR_INPUT
	uiNumber					: UINT;
END_VAR
//IF (__ISVALIDREF (THIS^.refstWybrana )) THEN
//	Zwroc 		:= THIS^.refstWybrana;
//END_IF
GetAdressOfRecipe			:= ADR (THIS^.arrRecipes [uiNumber]);
END_METHOD

(*			
	RafalOS
	Rafał Osajda		03.03.2025		TC 4026.13		wer. 0.0.0.1
	Zwraca referencje do  receptury
*)
METHOD PUBLIC GetChoosen : REFERENCE TO ST_BaseRecipe
//IF (__ISVALIDREF (THIS^.refstWybrana )) THEN
//	Zwroc 		:= THIS^.refstWybrana;
//END_IF
GetChoosen			REF= THIS^.GetReferenceToRecipe (uiNumer := THIS^.uiChosen);
END_METHOD

(*			
	RafalOS
	Rafał Osajda		03.03.2025		TC 4026.13		wer. 0.0.0.1
	
*)
METHOD PUBLIC GetIngredientFromRecipe : ST_BaseDescriptor
VAR_INPUT
	uiNumberOfRecipe			: UINT;
	uiNumberOfIngredient		: UINT;
END_VAR
GetIngredientFromRecipe			:= THIS^.arrRecipes [uiNumberOfRecipe].arrIngredient [uiNumberOfIngredient];
END_METHOD

(*			
	RafalOS
	Rafał Osajda		03.03.2025		TC 4026.13		wer. 0.0.0.1
	
*)
METHOD PUBLIC GetIngredientFromTemplate : ST_BaseDescriptor
VAR_INPUT
	uiNumberOfTemplate			: UINT;
	uiNumberOfIngredient		: UINT;
END_VAR
GetIngredientFromTemplate			:= THIS^.arrRecipes [uiNumberOfTemplate].arrIngredient [uiNumberOfIngredient];
END_METHOD

(*			
	RafalOS
	Rafał Osajda		02.12.2025		TC 4024.66
	Zwraca do tablicy wybrany zakres składników
*)
METHOD PUBLIC GetIngredientRange 
VAR_INPUT
	iRecipe			: INT;	//numer receptury z której bierzemy składniki
	iStartIndex		: INT;	//numer startowy składnika
	iCount			: INT;	//ilośc pobieranych 
END_VAR
VAR_IN_OUT
	arrOut : ARRAY [*] OF ST_BaseDescriptor;
END_VAR
VAR_OUTPUT
	iNumberOfFilledData	: INT;	//ilosc wypelnionych danych na strone
END_VAR
VAR
	itmpCount		: INT;
	iI				: INT;
	iJ				: INT;
	sttmpEmpty		: ST_BaseDescriptor;
END_VAR
itmpCount := iStartIndex + iCount - 2;
iJ := 0;
FOR iI := iStartIndex TO itmpCount DO
	IF (iI <= TO_INT (THIS^.arrRecipes [iRecipe].uiNumber)) THEN
		iJ := iJ + 1;
		arrOut [iJ] := THIS^.arrRecipes [iRecipe].arrIngredient [iI];
		
	ELSE
		arrOut [iI] := sttmpEmpty;
	END_IF
END_FOR
iNumberOfFilledData := iJ;
END_METHOD

METHOD GetNameList : ST_BaseRecipeList
VAR
	iI			: INT;
	stResult	: ST_BaseRecipeList;
END_VAR
FOR iI := 1 TO TO_INT (THIS^.uiNumberOfRecipes) DO
	stResult.arrName [iI] := THIS^.arrRecipes [iI].stTexts;
	stResult.iNumber := stResult.iNumber + 1;
END_FOR
GetNameList := stResult;
END_METHOD

METHOD GetNameListTemplate : ST_BaseRecipeList
VAR
	iI			: INT;
	stResult	: ST_BaseRecipeList;
END_VAR
FOR iI := 1 TO TO_INT (THIS^.uiNumberOfTemplates) DO
	stResult.arrName [iI] := THIS^.arrTemplates [iI].stTexts;
	stResult.iNumber := stResult.iNumber + 1;
END_FOR
GetNameListTemplate := stResult;
END_METHOD

METHOD GetNamesOfRecipe : ST_BaseLabel
VAR_INPUT
	uiNumber			: UINT;
END_VAR
GetNamesOfRecipe			:= THIS^.arrRecipes [uiNumber].stTexts;
END_METHOD

METHOD GetNamesOfSelectRecipe : ST_BaseLabel
VAR_INPUT

END_VAR
GetNamesOfSelectRecipe := THIS^.GetNamesOfRecipe (uiNumber := THIS^.uiChosen);
END_METHOD

METHOD PUBLIC GetNamesOfTemplate : ST_BaseLabel
VAR_INPUT
	uiNumber			: UINT;
END_VAR
GetNamesOfTemplate			:= THIS^.arrTemplates [uiNumber].stTexts;
END_METHOD

(*			
	RafalOS
	Rafał Osajda		03.03.2025		TC 4026.13		wer. 0.0.0.1
	
*)
METHOD PUBLIC GetNumberIngredientOfRecipe : UINT
VAR_INPUT
	uiNumber				: UINT;
END_VAR
GetNumberIngredientOfRecipe 		:= THIS^.arrRecipes [uiNumber].uiNumber;
END_METHOD

METHOD PUBLIC GetNumberIngredientOFTemplate : UINT
VAR_INPUT
	uiNumber				: UINT;
END_VAR
GetNumberIngredientOFTemplate 		:= THIS^.arrTemplates [uiNumber].uiNumber;
END_METHOD

METHOD PUBLIC GetNumberOfChoosen : UINT
VAR_INPUT
END_VAR
GetNumberOfChoosen			:= THIS^.uiChosen;
END_METHOD

METHOD PUBLIC GetNumberOfCreatingRecipe : UINT
VAR_INPUT
END_VAR
GetNumberOfCreatingRecipe := THIS^.uiNumberOfCreatingRecipe;
END_METHOD

METHOD PUBLIC GetNumberOfRecipe : UINT
VAR_INPUT
END_VAR
GetNumberOfRecipe			:= THIS^.uiNumberOfRecipes;
END_METHOD

METHOD PUBLIC GetNumberOfTemplate : UINT
VAR_INPUT
END_VAR
GetNumberOfTemplate		:= THIS^.uiNumberOfTemplates;
END_METHOD

